LIN {X 0,Y 354.82,Z 335.287,A -85,B 0,C 180,E1 -13355.7,E2 -13355.7} C_VEL
LIN {X 0,Y 354.766,Z 335.295,A -85,B 0,C 180,E1 -13359.413,E2 -13359.413} C_VEL
LIN {X 0,Y 354.779,Z 335.292,A -85,B 0,C 180,E1 -13362.866,E2 -13362.866} C_VEL
LIN {X 0,Y 354.841,Z 335.416,A -85,B 0,C 180,E1 -13366.284,E2 -13366.284} C_VEL
LIN {X 0,Y 355.568,Z 339.552,A -85,B 0,C 180,E1 -13369.288,E2 -13369.288} C_VEL
LIN {X 0,Y 356.215,Z 343.93,A -85,B 0,C 180,E1 -13372.294,E2 -13372.294} C_VEL
LIN {X 0,Y 356.345,Z 348.318,A -85,B 0,C 180,E1 -13375.114,E2 -13375.114} C_VEL
LIN {X 0,Y 355.9,Z 353.266,A -85,B 0,C 180,E1 -13378.117,E2 -13378.117} C_VEL
LIN {X 0,Y 355.284,Z 359.294,A -85,B 0,C 180,E1 -13381.657,E2 -13381.657} C_VEL
LIN {X 0,Y 354.717,Z 365.813,A -85,B 0,C 180,E1 -13385.413,E2 -13385.413} C_VEL
LIN {X 0,Y 354.237,Z 372.787,A -85,B 0,C 180,E1 -13389.381,E2 -13389.381} C_VEL
LIN {X 0,Y 354.223,Z 372.987,A -85,B 0,C 180,E1 -13389.494,E2 -13389.494} C_VEL
LIN {X 0,Y 357.148,Z 387.433,A -85,B 0,C 180,E1 -13390.215,E2 -13390.215} C_VEL
LIN {X 0,Y 359.09,Z 400.479,A -85,B 0,C 180,E1 -13391.066,E2 -13391.066} C_VEL
LIN {X 0,Y 360.005,Z 409.631,A -85,B 0,C 180,E1 -13391.799,E2 -13391.799} C_VEL
LIN {X 0,Y 358.951,Z 420.65,A -85,B 0,C 180,E1 -13392.774,E2 -13392.774} C_VEL
LIN {X 0,Y 357.794,Z 431.905,A -85,B 0,C 180,E1 -13394.038,E2 -13394.038} C_VEL
LIN {X 0,Y 356.687,Z 441.874,A -85,B 0,C 180,E1 -13395.45,E2 -13395.45} C_VEL
LIN {X 0,Y 355.611,Z 451.544,A -85,B 0,C 180,E1 -13397.154,E2 -13397.154} C_VEL
LIN {X 0,Y 354.701,Z 459.242,A -85,B 0,C 180,E1 -13398.861,E2 -13398.861} C_VEL
LIN {X 0,Y 353.989,Z 466.343,A -85,B 0,C 180,E1 -13400.861,E2 -13400.861} C_VEL
LIN {X 0,Y 353.617,Z 471.071,A -85,B 0,C 180,E1 -13402.577,E2 -13402.577} C_VEL
LIN {X 0,Y 353.338,Z 474.682,A -85,B 0,C 180,E1 -13404.292,E2 -13404.292} C_VEL
LIN {X 0,Y 353.3,Z 476.548,A -85,B 0,C 180,E1 -13405.436,E2 -13405.436} C_VEL
LIN {X 0,Y 353.226,Z 477.946,A -85,B 0,C 180,E1 -13406.578,E2 -13406.578} C_VEL
LIN {X 0,Y 353.194,Z 479.554,A -85,B 0,C 180,E1 -13408.859,E2 -13408.859} C_VEL
LIN {X 0,Y 353.218,Z 479.771,A -85,B 0,C 180,E1 -13409.999,E2 -13409.999} C_VEL
LIN {X 0,Y 353.194,Z 479.553,A -85,B 0,C 180,E1 -13411.14,E2 -13411.14} C_VEL
LIN {X 0,Y 353.225,Z 477.945,A -85,B 0,C 180,E1 -13413.421,E2 -13413.421} C_VEL
LIN {X 0,Y 353.299,Z 476.546,A -85,B 0,C 180,E1 -13414.563,E2 -13414.563} C_VEL
LIN {X 0,Y 353.388,Z 473.979,A -85,B 0,C 180,E1 -13416.079,E2 -13416.079} C_VEL
LIN {X 0,Y 353.694,Z 469.623,A -85,B 0,C 180,E1 -13417.995,E2 -13417.995} C_VEL
LIN {X 0,Y 354.271,Z 463.506,A -85,B 0,C 180,E1 -13419.995,E2 -13419.995} C_VEL
LIN {X 0,Y 354.957,Z 456.823,A -85,B 0,C 180,E1 -13421.709,E2 -13421.709} C_VEL
LIN {X 0,Y 355.974,Z 448.538,A -85,B 0,C 180,E1 -13423.413,E2 -13423.413} C_VEL
LIN {X 0,Y 356.928,Z 440.045,A -85,B 0,C 180,E1 -13424.83,E2 -13424.83} C_VEL
LIN {X 0,Y 357.971,Z 429.549,A -85,B 0,C 180,E1 -13426.246,E2 -13426.246} C_VEL
LIN {X 0,Y 359.253,Z 417.743,A -85,B 0,C 180,E1 -13427.503,E2 -13427.503} C_VEL
LIN {X 0,Y 359.988,Z 408.468,A -85,B 0,C 180,E1 -13428.292,E2 -13428.292} C_VEL
LIN {X 0,Y 358.547,Z 396.566,A -85,B 0,C 180,E1 -13429.209,E2 -13429.209} C_VEL
LIN {X 0,Y 356.404,Z 383.633,A -85,B 0,C 180,E1 -13429.988,E2 -13429.988} C_VEL
LIN {X 0,Y 354.221,Z 372.993,A -85,B 0,C 180,E1 -13430.495,E2 -13430.495} C_VEL
LIN {X 0,Y 354.745,Z 365.803,A -85,B 0,C 180,E1 -13434.584,E2 -13434.584} C_VEL
LIN {X 0,Y 355.28,Z 359.281,A -85,B 0,C 180,E1 -13438.342,E2 -13438.342} C_VEL
LIN {X 0,Y 355.955,Z 352.692,A -85,B 0,C 180,E1 -13442.213,E2 -13442.213} C_VEL
LIN {X 0,Y 356.359,Z 348.294,A -85,B 0,C 180,E1 -13444.883,E2 -13444.883} C_VEL
LIN {X 0,Y 356.219,Z 343.604,A -85,B 0,C 180,E1 -13447.891,E2 -13447.891} C_VEL
LIN {X 0,Y 355.485,Z 338.678,A -85,B 0,C 180,E1 -13451.3,E2 -13451.3} C_VEL
LIN {X 0,Y 354.865,Z 335.288,A -85,B 0,C 180,E1 -13453.879,E2 -13453.879} C_VEL
LIN {X 0,Y 354.783,Z 335.289,A -85,B 0,C 180,E1 -13457.661,E2 -13457.661} C_VEL
LIN {X 0,Y 354.778,Z 335.295,A -85,B 0,C 180,E1 -13460.661,E2 -13460.661} C_VEL
LIN {X 0,Y 354.815,Z 335.287,A -85,B 0,C 180,E1 -13464.3,E2 -13464.3} C_VEL
LIN {X 0,Y 354.779,Z 335.289,A -85,B 0,C 180,E1 -13467.666,E2 -13467.666} C_VEL
LIN {X 0,Y 354.792,Z 335.288,A -85,B 0,C 180,E1 -13471.614,E2 -13471.614} C_VEL
LIN {X 0,Y 354.826,Z 335.284,A -85,B 0,C 180,E1 -13475.656,E2 -13475.656} C_VEL
LIN {X 0,Y 354.818,Z 335.284,A -85,B 0,C 180,E1 -13479.113,E2 -13479.113} C_VEL
LIN {X 0,Y 354.889,Z 335.276,A -85,B 0,C 180,E1 -13482.719,E2 -13482.719} C_VEL
LIN {X 0,Y 354.942,Z 335.273,A -85,B 0,C 180,E1 -13486.255,E2 -13486.255} C_VEL
LIN {X 0,Y 354.968,Z 335.269,A -85,B 0,C 180,E1 -13489.736,E2 -13489.736} C_VEL
LIN {X 0,Y 355.105,Z 335.253,A -85,B 0,C 180,E1 -13492.037,E2 -13492.037} C_VEL
LIN {X 0,Y 355.089,Z 335.252,A -85,B 0,C 180,E1 -13494.321,E2 -13494.321} C_VEL
LIN {X 0,Y 355.236,Z 335.238,A -85,B 0,C 180,E1 -13497.732,E2 -13497.732} C_VEL
LIN {X 0,Y 355.302,Z 335.227,A -85,B 0,C 180,E1 -13500,E2 -13500} C_VEL
LIN {X 0,Y 355.234,Z 335.233,A -85,B 0,C 180,E1 -13502.268,E2 -13502.268} C_VEL
LIN {X 0,Y 355.129,Z 335.246,A -85,B 0,C 180,E1 -13506.819,E2 -13506.819} C_VEL
LIN {X 0,Y 355.006,Z 335.263,A -85,B 0,C 180,E1 -13509.113,E2 -13509.113} C_VEL
LIN {X 0,Y 354.912,Z 335.273,A -85,B 0,C 180,E1 -13512.581,E2 -13512.581} C_VEL
LIN {X 0,Y 354.88,Z 335.276,A -85,B 0,C 180,E1 -13516.097,E2 -13516.097} C_VEL
LIN {X 0,Y 354.893,Z 335.275,A -85,B 0,C 180,E1 -13518.473,E2 -13518.473} C_VEL
LIN {X 0,Y 354.822,Z 335.283,A -85,B 0,C 180,E1 -13522.107,E2 -13522.107} C_VEL
LIN {X 0,Y 354.807,Z 335.286,A -85,B 0,C 180,E1 -13525.835,E2 -13525.835} C_VEL
LIN {X 0,Y 354.789,Z 335.288,A -85,B 0,C 180,E1 -13529.685,E2 -13529.685} C_VEL
LIN {X 0,Y 354.78,Z 335.29,A -85,B 0,C 180,E1 -13532.334,E2 -13532.334} C_VEL
LIN {X 0,Y 354.815,Z 335.284,A -85,B 0,C 180,E1 -13535.7,E2 -13535.7} C_VEL
LIN {X 0,Y 354.762,Z 335.291,A -85,B 0,C 180,E1 -13539.413,E2 -13539.413} C_VEL
LIN {X 0,Y 354.779,Z 335.292,A -85,B 0,C 180,E1 -13542.868,E2 -13542.868} C_VEL
LIN {X 0,Y 354.771,Z 335.293,A -85,B 0,C 180,E1 -13546.106,E2 -13546.106} C_VEL
LIN {X 0,Y 354.821,Z 335.284,A -85,B 0,C 180,E1 -13549.185,E2 -13549.185} C_VEL
LIN {X 0,Y 354.775,Z 335.296,A -85,B 0,C 180,E1 -13552.41,E2 -13552.41} C_VEL
LIN {X 0,Y 354.745,Z 335.624,A -85,B 0,C 180,E1 -13553.536,E2 -13553.536} C_VEL
LIN {X 0,Y 354.755,Z 338.537,A -85,B 0,C 180,E1 -13556.311,E2 -13556.311} C_VEL
LIN {X 0,Y 354.589,Z 341.488,A -85,B 0,C 180,E1 -13558.982,E2 -13558.982} C_VEL
LIN {X 0,Y 354.382,Z 344.409,A -85,B 0,C 180,E1 -13561.579,E2 -13561.579} C_VEL
LIN {X 0,Y 354.195,Z 347.361,A -85,B 0,C 180,E1 -13564.119,E2 -13564.119} C_VEL
LIN {X 0,Y 354.058,Z 350.336,A -85,B 0,C 180,E1 -13566.61,E2 -13566.61} C_VEL
LIN {X 0,Y 353.917,Z 354.113,A -85,B 0,C 180,E1 -13569.579,E2 -13569.579} C_VEL
LIN {X 0,Y 357.383,Z 367.353,A -85,B 0,C 180,E1 -13570.301,E2 -13570.301} C_VEL
LIN {X 0,Y 360.021,Z 379.994,A -85,B 0,C 180,E1 -13571.183,E2 -13571.183} C_VEL
LIN {X 0,Y 360.821,Z 385.123,A -85,B 0,C 180,E1 -13571.598,E2 -13571.598} C_VEL
LIN {X 0,Y 359.833,Z 396.447,A -85,B 0,C 180,E1 -13572.526,E2 -13572.526} C_VEL
LIN {X 0,Y 358.761,Z 407.702,A -85,B 0,C 180,E1 -13573.719,E2 -13573.719} C_VEL
LIN {X 0,Y 357.883,Z 416.823,A -85,B 0,C 180,E1 -13574.919,E2 -13574.919} C_VEL
LIN {X 0,Y 356.769,Z 425.661,A -85,B 0,C 180,E1 -13576.327,E2 -13576.327} C_VEL
LIN {X 0,Y 355.762,Z 434.277,A -85,B 0,C 180,E1 -13578.029,E2 -13578.029} C_VEL
LIN {X 0,Y 354.929,Z 441.145,A -85,B 0,C 180,E1 -13579.735,E2 -13579.735} C_VEL
LIN {X 0,Y 354.244,Z 446.645,A -85,B 0,C 180,E1 -13581.444,E2 -13581.444} C_VEL
LIN {X 0,Y 353.809,Z 451.294,A -85,B 0,C 180,E1 -13583.312,E2 -13583.312} C_VEL
LIN {X 0,Y 353.502,Z 455.095,A -85,B 0,C 180,E1 -13585.439,E2 -13585.439} C_VEL
LIN {X 0,Y 353.343,Z 456.494,A -85,B 0,C 180,E1 -13586.58,E2 -13586.58} C_VEL
LIN {X 0,Y 353.271,Z 458.097,A -85,B 0,C 180,E1 -13588.861,E2 -13588.861} C_VEL
LIN {X 0,Y 353.266,Z 458.329,A -85,B 0,C 180,E1 -13590.001,E2 -13590.001} C_VEL
LIN {X 0,Y 353.271,Z 458.139,A -85,B 0,C 180,E1 -13591.14,E2 -13591.14} C_VEL
LIN {X 0,Y 353.341,Z 456.589,A -85,B 0,C 180,E1 -13593.421,E2 -13593.421} C_VEL
LIN {X 0,Y 353.499,Z 455.231,A -85,B 0,C 180,E1 -13594.562,E2 -13594.562} C_VEL
LIN {X 0,Y 353.749,Z 452.388,A -85,B 0,C 180,E1 -13596.262,E2 -13596.262} C_VEL
LIN {X 0,Y 354.072,Z 448.483,A -85,B 0,C 180,E1 -13597.987,E2 -13597.987} C_VEL
LIN {X 0,Y 354.642,Z 443.469,A -85,B 0,C 180,E1 -13599.698,E2 -13599.698} C_VEL
LIN {X 0,Y 355.378,Z 437.156,A -85,B 0,C 180,E1 -13601.406,E2 -13601.406} C_VEL
LIN {X 0,Y 356.349,Z 429.251,A -85,B 0,C 180,E1 -13603.109,E2 -13603.109} C_VEL
LIN {X 0,Y 357.586,Z 419.416,A -85,B 0,C 180,E1 -13604.804,E2 -13604.804} C_VEL
LIN {X 0,Y 358.586,Z 409.357,A -85,B 0,C 180,E1 -13606.185,E2 -13606.185} C_VEL
LIN {X 0,Y 359.604,Z 398.868,A -85,B 0,C 180,E1 -13607.34,E2 -13607.34} C_VEL
LIN {X 0,Y 360.695,Z 387.231,A -85,B 0,C 180,E1 -13608.349,E2 -13608.349} C_VEL
LIN {X 0,Y 360.661,Z 383.615,A -85,B 0,C 180,E1 -13608.626,E2 -13608.626} C_VEL
LIN {X 0,Y 358.538,Z 372.554,A -85,B 0,C 180,E1 -13609.465,E2 -13609.465} C_VEL
LIN {X 0,Y 355.39,Z 359.719,A -85,B 0,C 180,E1 -13610.251,E2 -13610.251} C_VEL
LIN {X 0,Y 353.911,Z 353.989,A -85,B 0,C 180,E1 -13610.555,E2 -13610.555} C_VEL
LIN {X 0,Y 354.113,Z 348.985,A -85,B 0,C 180,E1 -13614.632,E2 -13614.632} C_VEL
LIN {X 0,Y 354.299,Z 346.026,A -85,B 0,C 180,E1 -13617.144,E2 -13617.144} C_VEL
LIN {X 0,Y 354.588,Z 341.593,A -85,B 0,C 180,E1 -13621.019,E2 -13621.019} C_VEL
LIN {X 0,Y 354.758,Z 338.678,A -85,B 0,C 180,E1 -13623.69,E2 -13623.69} C_VEL
LIN {X 0,Y 354.749,Z 335.746,A -85,B 0,C 180,E1 -13626.465,E2 -13626.465} C_VEL
LIN {X 0,Y 354.785,Z 335.294,A -85,B 0,C 180,E1 -13627.868,E2 -13627.868} C_VEL
LIN {X 0,Y 354.143,Z 335.374,A -85,B 0,C 180,E1 -13628.815,E2 -13628.815} C_VEL
LIN {X 0,Y 351.27,Z 335.728,A -85,B 0,C 180,E1 -13630.354,E2 -13630.354} C_VEL
LIN {X 0,Y 348.826,Z 336.037,A -85,B 0,C 180,E1 -13631.6,E2 -13631.6} C_VEL
LIN {X 0,Y 347.786,Z 336.161,A -85,B 0,C 180,E1 -13632.564,E2 -13632.564} C_VEL
LIN {X 0,Y 347.709,Z 336.171,A -85,B 0,C 180,E1 -13632.891,E2 -13632.891} C_VEL
LIN {X 0,Y 347.721,Z 336.169,A -85,B 0,C 180,E1 -13636.687,E2 -13636.687} C_VEL
LIN {X 0,Y 347.699,Z 336.171,A -85,B 0,C 180,E1 -13640.182,E2 -13640.182} C_VEL
LIN {X 0,Y 347.755,Z 336.164,A -85,B 0,C 180,E1 -13642.678,E2 -13642.678} C_VEL
LIN {X 0,Y 347.747,Z 336.166,A -85,B 0,C 180,E1 -13645.956,E2 -13645.956} C_VEL
LIN {X 0,Y 347.736,Z 336.168,A -85,B 0,C 180,E1 -13649.651,E2 -13649.651} C_VEL
LIN {X 0,Y 347.746,Z 336.166,A -85,B 0,C 180,E1 -13653.601,E2 -13653.601} C_VEL
LIN {X 0,Y 347.767,Z 336.162,A -85,B 0,C 180,E1 -13656.16,E2 -13656.16} C_VEL
LIN {X 0,Y 347.804,Z 336.158,A -85,B 0,C 180,E1 -13659.909,E2 -13659.909} C_VEL
LIN {X 0,Y 347.863,Z 336.152,A -85,B 0,C 180,E1 -13662.359,E2 -13662.359} C_VEL
LIN {X 0,Y 347.895,Z 336.147,A -85,B 0,C 180,E1 -13665.971,E2 -13665.971} C_VEL
LIN {X 0,Y 347.925,Z 336.143,A -85,B 0,C 180,E1 -13669.525,E2 -13669.525} C_VEL
LIN {X 0,Y 348.105,Z 336.122,A -85,B 0,C 180,E1 -13673.042,E2 -13673.042} C_VEL
LIN {X 0,Y 348.202,Z 336.109,A -85,B 0,C 180,E1 -13677.686,E2 -13677.686} C_VEL
LIN {X 0,Y 348.258,Z 336.104,A -85,B 0,C 180,E1 -13680,E2 -13680} C_VEL
LIN {X 0,Y 348.202,Z 336.114,A -85,B 0,C 180,E1 -13682.313,E2 -13682.313} C_VEL
LIN {X 0,Y 348.089,Z 336.123,A -85,B 0,C 180,E1 -13686.958,E2 -13686.958} C_VEL
LIN {X 0,Y 347.925,Z 336.145,A -85,B 0,C 180,E1 -13690.474,E2 -13690.474} C_VEL
LIN {X 0,Y 347.896,Z 336.151,A -85,B 0,C 180,E1 -13694.15,E2 -13694.15} C_VEL
LIN {X 0,Y 347.888,Z 336.15,A -85,B 0,C 180,E1 -13698.29,E2 -13698.29} C_VEL
LIN {X 0,Y 347.773,Z 336.167,A -85,B 0,C 180,E1 -13701.63,E2 -13701.63} C_VEL
LIN {X 0,Y 347.766,Z 336.164,A -85,B 0,C 180,E1 -13705.112,E2 -13705.112} C_VEL
LIN {X 0,Y 347.734,Z 336.172,A -85,B 0,C 180,E1 -13707.701,E2 -13707.701} C_VEL
LIN {X 0,Y 347.736,Z 336.167,A -85,B 0,C 180,E1 -13710.349,E2 -13710.349} C_VEL
LIN {X 0,Y 347.747,Z 336.166,A -85,B 0,C 180,E1 -13714.044,E2 -13714.044} C_VEL
LIN {X 0,Y 347.755,Z 336.17,A -85,B 0,C 180,E1 -13717.322,E2 -13717.322} C_VEL
LIN {X 0,Y 347.736,Z 336.169,A -85,B 0,C 180,E1 -13721.601,E2 -13721.601} C_VEL
LIN {X 0,Y 347.722,Z 336.173,A -85,B 0,C 180,E1 -13725.431,E2 -13725.431} C_VEL
LIN {X 0,Y 347.746,Z 336.196,A -85,B 0,C 180,E1 -13725.836,E2 -13725.836} C_VEL
LIN {X 0,Y 348.543,Z 340.513,A -85,B 0,C 180,E1 -13729.07,E2 -13729.07} C_VEL
LIN {X 0,Y 349.123,Z 344.279,A -85,B 0,C 180,E1 -13731.729,E2 -13731.729} C_VEL
LIN {X 0,Y 349.343,Z 348.156,A -85,B 0,C 180,E1 -13734.309,E2 -13734.309} C_VEL
LIN {X 0,Y 349.062,Z 352.543,A -85,B 0,C 180,E1 -13737.07,E2 -13737.07} C_VEL
LIN {X 0,Y 348.484,Z 357.61,A -85,B 0,C 180,E1 -13740.135,E2 -13740.135} C_VEL
LIN {X 0,Y 347.913,Z 363.445,A -85,B 0,C 180,E1 -13743.614,E2 -13743.614} C_VEL
LIN {X 0,Y 347.384,Z 369.908,A -85,B 0,C 180,E1 -13747.394,E2 -13747.394} C_VEL
LIN {X 0,Y 347.233,Z 372.918,A -85,B 0,C 180,E1 -13749.081,E2 -13749.081} C_VEL
LIN {X 0,Y 349.979,Z 386.18,A -85,B 0,C 180,E1 -13749.741,E2 -13749.741} C_VEL
LIN {X 0,Y 352.067,Z 399.457,A -85,B 0,C 180,E1 -13750.62,E2 -13750.62} C_VEL
LIN {X 0,Y 353.173,Z 409.418,A -85,B 0,C 180,E1 -13751.434,E2 -13751.434} C_VEL
LIN {X 0,Y 352.175,Z 420.438,A -85,B 0,C 180,E1 -13752.432,E2 -13752.432} C_VEL
LIN {X 0,Y 350.947,Z 431.692,A -85,B 0,C 180,E1 -13753.718,E2 -13753.718} C_VEL
LIN {X 0,Y 349.806,Z 441.661,A -85,B 0,C 180,E1 -13755.157,E2 -13755.157} C_VEL
LIN {X 0,Y 348.654,Z 451.33,A -85,B 0,C 180,E1 -13756.893,E2 -13756.893} C_VEL
LIN {X 0,Y 347.698,Z 459.027,A -85,B 0,C 180,E1 -13758.634,E2 -13758.634} C_VEL
LIN {X 0,Y 346.95,Z 466.128,A -85,B 0,C 180,E1 -13760.674,E2 -13760.674} C_VEL
LIN {X 0,Y 346.542,Z 470.855,A -85,B 0,C 180,E1 -13762.425,E2 -13762.425} C_VEL
LIN {X 0,Y 346.27,Z 474.467,A -85,B 0,C 180,E1 -13764.175,E2 -13764.175} C_VEL
LIN {X 0,Y 346.216,Z 476.333,A -85,B 0,C 180,E1 -13765.342,E2 -13765.342} C_VEL
LIN {X 0,Y 346.15,Z 477.731,A -85,B 0,C 180,E1 -13766.508,E2 -13766.508} C_VEL
LIN {X 0,Y 346.095,Z 479.338,A -85,B 0,C 180,E1 -13768.836,E2 -13768.836} C_VEL
LIN {X 0,Y 346.121,Z 479.556,A -85,B 0,C 180,E1 -13769.999,E2 -13769.999} C_VEL
LIN {X 0,Y 346.095,Z 479.337,A -85,B 0,C 180,E1 -13771.163,E2 -13771.163} C_VEL
LIN {X 0,Y 346.15,Z 477.73,A -85,B 0,C 180,E1 -13773.491,E2 -13773.491} C_VEL
LIN {X 0,Y 346.215,Z 476.33,A -85,B 0,C 180,E1 -13774.657,E2 -13774.657} C_VEL
LIN {X 0,Y 346.279,Z 474.111,A -85,B 0,C 180,E1 -13776.014,E2 -13776.014} C_VEL
LIN {X 0,Y 346.646,Z 469.406,A -85,B 0,C 180,E1 -13778.158,E2 -13778.158} C_VEL
LIN {X 0,Y 347.256,Z 463.289,A -85,B 0,C 180,E1 -13780.199,E2 -13780.199} C_VEL
LIN {X 0,Y 347.987,Z 456.606,A -85,B 0,C 180,E1 -13781.946,E2 -13781.946} C_VEL
LIN {X 0,Y 349.05,Z 448.32,A -85,B 0,C 180,E1 -13783.684,E2 -13783.684} C_VEL
LIN {X 0,Y 350.04,Z 439.826,A -85,B 0,C 180,E1 -13785.129,E2 -13785.129} C_VEL
LIN {X 0,Y 351.127,Z 429.329,A -85,B 0,C 180,E1 -13786.571,E2 -13786.571} C_VEL
LIN {X 0,Y 352.316,Z 418.952,A -85,B 0,C 180,E1 -13787.71,E2 -13787.71} C_VEL
LIN {X 0,Y 353.114,Z 409.34,A -85,B 0,C 180,E1 -13788.568,E2 -13788.568} C_VEL
LIN {X 0,Y 351.771,Z 397.659,A -85,B 0,C 180,E1 -13789.508,E2 -13789.508} C_VEL
LIN {X 0,Y 349.728,Z 385.039,A -85,B 0,C 180,E1 -13790.318,E2 -13790.318} C_VEL
LIN {X 0,Y 347.207,Z 372.784,A -85,B 0,C 180,E1 -13790.92,E2 -13790.92} C_VEL
LIN {X 0,Y 347.667,Z 366.586,A -85,B 0,C 180,E1 -13794.541,E2 -13794.541} C_VEL
LIN {X 0,Y 348.24,Z 360.184,A -85,B 0,C 180,E1 -13798.31,E2 -13798.31} C_VEL
LIN {X 0,Y 348.91,Z 353.676,A -85,B 0,C 180,E1 -13802.221,E2 -13802.221} C_VEL
LIN {X 0,Y 349.353,Z 349.215,A -85,B 0,C 180,E1 -13804.983,E2 -13804.983} C_VEL
LIN {X 0,Y 349.303,Z 345.922,A -85,B 0,C 180,E1 -13807.127,E2 -13807.127} C_VEL
LIN {X 0,Y 348.759,Z 341.553,A -85,B 0,C 180,E1 -13810.153,E2 -13810.153} C_VEL
LIN {X 0,Y 347.938,Z 336.657,A -85,B 0,C 180,E1 -13813.771,E2 -13813.771} C_VEL
LIN {X 0,Y 347.839,Z 336.164,A -85,B 0,C 180,E1 -13814.17,E2 -13814.17} C_VEL
LIN {X 0,Y 347.735,Z 336.17,A -85,B 0,C 180,E1 -13818.398,E2 -13818.398} C_VEL
LIN {X 0,Y 347.751,Z 336.17,A -85,B 0,C 180,E1 -13822.678,E2 -13822.678} C_VEL
LIN {X 0,Y 347.741,Z 336.167,A -85,B 0,C 180,E1 -13825.955,E2 -13825.955} C_VEL
LIN {X 0,Y 347.73,Z 336.167,A -85,B 0,C 180,E1 -13829.65,E2 -13829.65} C_VEL
LIN {X 0,Y 347.741,Z 336.166,A -85,B 0,C 180,E1 -13833.6,E2 -13833.6} C_VEL
LIN {X 0,Y 347.762,Z 336.168,A -85,B 0,C 180,E1 -13836.16,E2 -13836.16} C_VEL
LIN {X 0,Y 347.798,Z 336.161,A -85,B 0,C 180,E1 -13839.908,E2 -13839.908} C_VEL
LIN {X 0,Y 347.857,Z 336.155,A -85,B 0,C 180,E1 -13842.359,E2 -13842.359} C_VEL
LIN {X 0,Y 347.889,Z 336.152,A -85,B 0,C 180,E1 -13845.97,E2 -13845.97} C_VEL
LIN {X 0,Y 347.919,Z 336.145,A -85,B 0,C 180,E1 -13849.525,E2 -13849.525} C_VEL
LIN {X 0,Y 348.066,Z 336.131,A -85,B 0,C 180,E1 -13851.875,E2 -13851.875} C_VEL
LIN {X 0,Y 348.064,Z 336.128,A -85,B 0,C 180,E1 -13854.206,E2 -13854.206} C_VEL
LIN {X 0,Y 348.199,Z 336.114,A -85,B 0,C 180,E1 -13857.687,E2 -13857.687} C_VEL
LIN {X 0,Y 348.254,Z 336.105,A -85,B 0,C 180,E1 -13860,E2 -13860} C_VEL
LIN {X 0,Y 348.197,Z 336.109,A -85,B 0,C 180,E1 -13862.314,E2 -13862.314} C_VEL
LIN {X 0,Y 348.099,Z 336.122,A -85,B 0,C 180,E1 -13866.958,E2 -13866.958} C_VEL
LIN {X 0,Y 347.919,Z 336.143,A -85,B 0,C 180,E1 -13870.475,E2 -13870.475} C_VEL
LIN {X 0,Y 347.89,Z 336.147,A -85,B 0,C 180,E1 -13874.15,E2 -13874.15} C_VEL
LIN {X 0,Y 347.882,Z 336.148,A -85,B 0,C 180,E1 -13878.291,E2 -13878.291} C_VEL
LIN {X 0,Y 347.778,Z 336.162,A -85,B 0,C 180,E1 -13881.635,E2 -13881.635} C_VEL
LIN {X 0,Y 347.761,Z 336.168,A -85,B 0,C 180,E1 -13885.113,E2 -13885.113} C_VEL
LIN {X 0,Y 347.728,Z 336.168,A -85,B 0,C 180,E1 -13887.701,E2 -13887.701} C_VEL
LIN {X 0,Y 347.731,Z 336.168,A -85,B 0,C 180,E1 -13890.35,E2 -13890.35} C_VEL
LIN {X 0,Y 347.742,Z 336.166,A -85,B 0,C 180,E1 -13894.045,E2 -13894.045} C_VEL
LIN {X 0,Y 347.75,Z 336.165,A -85,B 0,C 180,E1 -13897.322,E2 -13897.322} C_VEL
LIN {X 0,Y 347.735,Z 336.166,A -85,B 0,C 180,E1 -13901.602,E2 -13901.602} C_VEL
LIN {X 0,Y 347.702,Z 336.172,A -85,B 0,C 180,E1 -13905.028,E2 -13905.028} C_VEL
LIN {X 0,Y 347.764,Z 336.169,A -85,B 0,C 180,E1 -13908.395,E2 -13908.395} C_VEL
LIN {X 0,Y 347.755,Z 336.168,A -85,B 0,C 180,E1 -13912.016,E2 -13912.016} C_VEL
LIN {X 0,Y 347.702,Z 336.177,A -85,B 0,C 180,E1 -13912.673,E2 -13912.673} C_VEL
LIN {X 0,Y 347.746,Z 337.271,A -85,B 0,C 180,E1 -13914.121,E2 -13914.121} C_VEL
LIN {X 0,Y 347.659,Z 340.184,A -85,B 0,C 180,E1 -13916.921,E2 -13916.921} C_VEL
LIN {X 0,Y 347.427,Z 344.024,A -85,B 0,C 180,E1 -13920.44,E2 -13920.44} C_VEL
LIN {X 0,Y 347.203,Z 347.559,A -85,B 0,C 180,E1 -13923.557,E2 -13923.557} C_VEL
LIN {X 0,Y 347.06,Z 350.542,A -85,B 0,C 180,E1 -13926.11,E2 -13926.11} C_VEL
LIN {X 0,Y 346.864,Z 354.22,A -85,B 0,C 180,E1 -13929.132,E2 -13929.132} C_VEL
LIN {X 0,Y 350.573,Z 368.215,A -85,B 0,C 180,E1 -13929.933,E2 -13929.933} C_VEL
LIN {X 0,Y 353.168,Z 380.907,A -85,B 0,C 180,E1 -13930.85,E2 -13930.85} C_VEL
LIN {X 0,Y 353.995,Z 386.567,A -85,B 0,C 180,E1 -13931.323,E2 -13931.323} C_VEL
LIN {X 0,Y 352.919,Z 398.107,A -85,B 0,C 180,E1 -13932.322,E2 -13932.322} C_VEL
LIN {X 0,Y 351.892,Z 408.521,A -85,B 0,C 180,E1 -13933.468,E2 -13933.468} C_VEL
LIN {X 0,Y 351.051,Z 417.041,A -85,B 0,C 180,E1 -13934.618,E2 -13934.618} C_VEL
LIN {X 0,Y 349.889,Z 425.879,A -85,B 0,C 180,E1 -13936.053,E2 -13936.053} C_VEL
LIN {X 0,Y 348.828,Z 434.495,A -85,B 0,C 180,E1 -13937.788,E2 -13937.788} C_VEL
LIN {X 0,Y 347.957,Z 441.362,A -85,B 0,C 180,E1 -13939.527,E2 -13939.527} C_VEL
LIN {X 0,Y 347.232,Z 446.861,A -85,B 0,C 180,E1 -13941.269,E2 -13941.269} C_VEL
LIN {X 0,Y 346.731,Z 451.805,A -85,B 0,C 180,E1 -13943.315,E2 -13943.315} C_VEL
LIN {X 0,Y 346.443,Z 455.311,A -85,B 0,C 180,E1 -13945.346,E2 -13945.346} C_VEL
LIN {X 0,Y 346.267,Z 456.709,A -85,B 0,C 180,E1 -13946.51,E2 -13946.51} C_VEL
LIN {X 0,Y 346.175,Z 458.313,A -85,B 0,C 180,E1 -13948.837,E2 -13948.837} C_VEL
LIN {X 0,Y 346.17,Z 458.544,A -85,B 0,C 180,E1 -13950.001,E2 -13950.001} C_VEL
LIN {X 0,Y 346.175,Z 458.354,A -85,B 0,C 180,E1 -13951.164,E2 -13951.164} C_VEL
LIN {X 0,Y 346.266,Z 456.803,A -85,B 0,C 180,E1 -13953.491,E2 -13953.491} C_VEL
LIN {X 0,Y 346.441,Z 455.446,A -85,B 0,C 180,E1 -13954.655,E2 -13954.655} C_VEL
LIN {X 0,Y 346.795,Z 451.829,A -85,B 0,C 180,E1 -13956.774,E2 -13956.774} C_VEL
LIN {X 0,Y 347.189,Z 447.141,A -85,B 0,C 180,E1 -13958.733,E2 -13958.733} C_VEL
LIN {X 0,Y 348.023,Z 440.705,A -85,B 0,C 180,E1 -13960.766,E2 -13960.766} C_VEL
LIN {X 0,Y 348.891,Z 433.632,A -85,B 0,C 180,E1 -13962.507,E2 -13962.507} C_VEL
LIN {X 0,Y 350.062,Z 424.816,A -85,B 0,C 180,E1 -13964.237,E2 -13964.237} C_VEL
LIN {X 0,Y 351.218,Z 415.868,A -85,B 0,C 180,E1 -13965.657,E2 -13965.657} C_VEL
LIN {X 0,Y 352.132,Z 406.131,A -85,B 0,C 180,E1 -13966.927,E2 -13966.927} C_VEL
LIN {X 0,Y 353.321,Z 394.598,A -85,B 0,C 180,E1 -13968.108,E2 -13968.108} C_VEL
LIN {X 0,Y 353.957,Z 385.341,A -85,B 0,C 180,E1 -13968.877,E2 -13968.877} C_VEL
LIN {X 0,Y 351.567,Z 372.769,A -85,B 0,C 180,E1 -13969.867,E2 -13969.867} C_VEL
LIN {X 0,Y 348.465,Z 360.116,A -85,B 0,C 180,E1 -13970.665,E2 -13970.665} C_VEL
LIN {X 0,Y 346.847,Z 354.189,A -85,B 0,C 180,E1 -13971.002,E2 -13971.002} C_VEL
LIN {X 0,Y 347.041,Z 350.179,A -85,B 0,C 180,E1 -13974.313,E2 -13974.313} C_VEL
LIN {X 0,Y 347.287,Z 346.222,A -85,B 0,C 180,E1 -13977.739,E2 -13977.739} C_VEL
LIN {X 0,Y 347.603,Z 341.78,A -85,B 0,C 180,E1 -13981.714,E2 -13981.714} C_VEL
LIN {X 0,Y 347.744,Z 338.839,A -85,B 0,C 180,E1 -13984.464,E2 -13984.464} C_VEL
LIN {X 0,Y 347.758,Z 337.181,A -85,B 0,C 180,E1 -13986.062,E2 -13986.062} C_VEL
LIN {X 0,Y 347.702,Z 336.177,A -85,B 0,C 180,E1 -13987.328,E2 -13987.328} C_VEL
LIN {X 0,Y 347.732,Z 336.169,A -85,B 0,C 180,E1 -13990.297,E2 -13990.297} C_VEL
LIN {X 0,Y 347.709,Z 336.171,A -85,B 0,C 180,E1 -13992.891,E2 -13992.891} C_VEL
LIN {X 0,Y 347.069,Z 336.255,A -85,B 0,C 180,E1 -13993.858,E2 -13993.858} C_VEL
LIN {X 0,Y 344.257,Z 336.608,A -85,B 0,C 180,E1 -13995.432,E2 -13995.432} C_VEL
LIN {X 0,Y 341.844,Z 336.908,A -85,B 0,C 180,E1 -13996.706,E2 -13996.706} C_VEL
LIN {X 0,Y 340.784,Z 337.037,A -85,B 0,C 180,E1 -13997.691,E2 -13997.691} C_VEL
LIN {X 0,Y 340.684,Z 337.046,A -85,B 0,C 180,E1 -13998.025,E2 -13998.025} C_VEL
LIN {X 0,Y 340.718,Z 337.043,A -85,B 0,C 180,E1 -14001.77,E2 -14001.77} C_VEL
LIN {X 0,Y 340.722,Z 337.043,A -85,B 0,C 180,E1 -14005.595,E2 -14005.595} C_VEL
LIN {X 0,Y 340.691,Z 337.047,A -85,B 0,C 180,E1 -14008.954,E2 -14008.954} C_VEL
LIN {X 0,Y 340.717,Z 337.046,A -85,B 0,C 180,E1 -14013.012,E2 -14013.012} C_VEL
LIN {X 0,Y 340.739,Z 337.039,A -85,B 0,C 180,E1 -14015.637,E2 -14015.637} C_VEL
LIN {X 0,Y 340.732,Z 337.04,A -85,B 0,C 180,E1 -14019.473,E2 -14019.473} C_VEL
LIN {X 0,Y 340.855,Z 337.024,A -85,B 0,C 180,E1 -14021.984,E2 -14021.984} C_VEL
LIN {X 0,Y 340.867,Z 337.022,A -85,B 0,C 180,E1 -14025.705,E2 -14025.705} C_VEL
LIN {X 0,Y 340.868,Z 337.023,A -85,B 0,C 180,E1 -14029.306,E2 -14029.306} C_VEL
LIN {X 0,Y 341.075,Z 336.999,A -85,B 0,C 180,E1 -14032.898,E2 -14032.898} C_VEL
LIN {X 0,Y 341.164,Z 336.985,A -85,B 0,C 180,E1 -14037.639,E2 -14037.639} C_VEL
LIN {X 0,Y 341.211,Z 336.982,A -85,B 0,C 180,E1 -14040,E2 -14040} C_VEL
LIN {X 0,Y 341.163,Z 336.99,A -85,B 0,C 180,E1 -14042.361,E2 -14042.361} C_VEL
LIN {X 0,Y 341.057,Z 336.999,A -85,B 0,C 180,E1 -14047.102,E2 -14047.102} C_VEL
LIN {X 0,Y 340.868,Z 337.023,A -85,B 0,C 180,E1 -14050.694,E2 -14050.694} C_VEL
LIN {X 0,Y 340.86,Z 337.026,A -85,B 0,C 180,E1 -14054.325,E2 -14054.325} C_VEL
LIN {X 0,Y 340.834,Z 337.027,A -85,B 0,C 180,E1 -14058.466,E2 -14058.466} C_VEL
LIN {X 0,Y 340.718,Z 337.046,A -85,B 0,C 180,E1 -14061.843,E2 -14061.843} C_VEL
LIN {X 0,Y 340.717,Z 337.046,A -85,B 0,C 180,E1 -14065.669,E2 -14065.669} C_VEL
LIN {X 0,Y 340.703,Z 337.048,A -85,B 0,C 180,E1 -14069.674,E2 -14069.674} C_VEL
LIN {X 0,Y 340.684,Z 337.045,A -85,B 0,C 180,E1 -14072.436,E2 -14072.436} C_VEL
LIN {X 0,Y 340.716,Z 337.047,A -85,B 0,C 180,E1 -14075.279,E2 -14075.279} C_VEL
LIN {X 0,Y 340.692,Z 337.045,A -85,B 0,C 180,E1 -14078.383,E2 -14078.383} C_VEL
LIN {X 0,Y 340.689,Z 337.045,A -85,B 0,C 180,E1 -14082.044,E2 -14082.044} C_VEL
LIN {X 0,Y 340.71,Z 337.085,A -85,B 0,C 180,E1 -14085.466,E2 -14085.466} C_VEL
LIN {X 0,Y 341.493,Z 341.448,A -85,B 0,C 180,E1 -14088.81,E2 -14088.81} C_VEL
LIN {X 0,Y 342.148,Z 345.822,A -85,B 0,C 180,E1 -14091.959,E2 -14091.959} C_VEL
LIN {X 0,Y 342.328,Z 350.201,A -85,B 0,C 180,E1 -14094.912,E2 -14094.912} C_VEL
LIN {X 0,Y 341.774,Z 355.666,A -85,B 0,C 180,E1 -14098.375,E2 -14098.375} C_VEL
LIN {X 0,Y 341.059,Z 362.18,A -85,B 0,C 180,E1 -14102.384,E2 -14102.384} C_VEL
LIN {X 0,Y 340.449,Z 368.636,A -85,B 0,C 180,E1 -14106.263,E2 -14106.263} C_VEL
LIN {X 0,Y 340.192,Z 372.777,A -85,B 0,C 180,E1 -14108.629,E2 -14108.629} C_VEL
LIN {X 0,Y 342.938,Z 385.687,A -85,B 0,C 180,E1 -14109.292,E2 -14109.292} C_VEL
LIN {X 0,Y 344.93,Z 398.233,A -85,B 0,C 180,E1 -14110.134,E2 -14110.134} C_VEL
LIN {X 0,Y 346.188,Z 409.199,A -85,B 0,C 180,E1 -14111.045,E2 -14111.045} C_VEL
LIN {X 0,Y 345.902,Z 415.833,A -85,B 0,C 180,E1 -14111.643,E2 -14111.643} C_VEL
LIN {X 0,Y 344.648,Z 426.811,A -85,B 0,C 180,E1 -14112.801,E2 -14112.801} C_VEL
LIN {X 0,Y 343.44,Z 437.284,A -85,B 0,C 180,E1 -14114.203,E2 -14114.203} C_VEL
LIN {X 0,Y 342.284,Z 446.548,A -85,B 0,C 180,E1 -14115.736,E2 -14115.736} C_VEL
LIN {X 0,Y 341.146,Z 455.176,A -85,B 0,C 180,E1 -14117.507,E2 -14117.507} C_VEL
LIN {X 0,Y 340.359,Z 462.078,A -85,B 0,C 180,E1 -14119.29,E2 -14119.29} C_VEL
LIN {X 0,Y 339.741,Z 467.611,A -85,B 0,C 180,E1 -14121.074,E2 -14121.074} C_VEL
LIN {X 0,Y 339.367,Z 471.953,A -85,B 0,C 180,E1 -14122.862,E2 -14122.862} C_VEL
LIN {X 0,Y 339.19,Z 474.252,A -85,B 0,C 180,E1 -14124.053,E2 -14124.053} C_VEL
LIN {X 0,Y 339.118,Z 476.118,A -85,B 0,C 180,E1 -14125.244,E2 -14125.244} C_VEL
LIN {X 0,Y 339.077,Z 477.517,A -85,B 0,C 180,E1 -14126.435,E2 -14126.435} C_VEL
LIN {X 0,Y 338.998,Z 479.123,A -85,B 0,C 180,E1 -14128.812,E2 -14128.812} C_VEL
LIN {X 0,Y 339.025,Z 479.34,A -85,B 0,C 180,E1 -14129.999,E2 -14129.999} C_VEL
LIN {X 0,Y 338.998,Z 479.121,A -85,B 0,C 180,E1 -14131.187,E2 -14131.187} C_VEL
LIN {X 0,Y 339.077,Z 477.514,A -85,B 0,C 180,E1 -14133.564,E2 -14133.564} C_VEL
LIN {X 0,Y 339.115,Z 476.113,A -85,B 0,C 180,E1 -14134.755,E2 -14134.755} C_VEL
LIN {X 0,Y 339.25,Z 473.169,A -85,B 0,C 180,E1 -14136.542,E2 -14136.542} C_VEL
LIN {X 0,Y 339.591,Z 469.189,A -85,B 0,C 180,E1 -14138.329,E2 -14138.329} C_VEL
LIN {X 0,Y 340.233,Z 463.07,A -85,B 0,C 180,E1 -14140.412,E2 -14140.412} C_VEL
LIN {X 0,Y 341.014,Z 456.387,A -85,B 0,C 180,E1 -14142.194,E2 -14142.194} C_VEL
LIN {X 0,Y 342.133,Z 448.102,A -85,B 0,C 180,E1 -14143.966,E2 -14143.966} C_VEL
LIN {X 0,Y 343.275,Z 438.439,A -85,B 0,C 180,E1 -14145.617,E2 -14145.617} C_VEL
LIN {X 0,Y 344.445,Z 427.932,A -85,B 0,C 180,E1 -14147.055,E2 -14147.055} C_VEL
LIN {X 0,Y 345.704,Z 417.303,A -85,B 0,C 180,E1 -14148.213,E2 -14148.213} C_VEL
LIN {X 0,Y 346.301,Z 410.893,A -85,B 0,C 180,E1 -14148.794,E2 -14148.794} C_VEL
LIN {X 0,Y 345.086,Z 399.377,A -85,B 0,C 180,E1 -14149.769,E2 -14149.769} C_VEL
LIN {X 0,Y 343.087,Z 386.647,A -85,B 0,C 180,E1 -14150.64,E2 -14150.64} C_VEL
LIN {X 0,Y 340.434,Z 374.179,A -85,B 0,C 180,E1 -14151.306,E2 -14151.306} C_VEL
LIN {X 0,Y 340.174,Z 372.483,A -85,B 0,C 180,E1 -14151.423,E2 -14151.423} C_VEL
LIN {X 0,Y 340.621,Z 366.87,A -85,B 0,C 180,E1 -14154.79,E2 -14154.79} C_VEL
LIN {X 0,Y 341.185,Z 361.086,A -85,B 0,C 180,E1 -14158.278,E2 -14158.278} C_VEL
LIN {X 0,Y 341.764,Z 355.642,A -85,B 0,C 180,E1 -14161.625,E2 -14161.625} C_VEL
LIN {X 0,Y 342.329,Z 350.153,A -85,B 0,C 180,E1 -14165.087,E2 -14165.087} C_VEL
LIN {X 0,Y 342.155,Z 345.758,A -85,B 0,C 180,E1 -14168.038,E2 -14168.038} C_VEL
LIN {X 0,Y 341.542,Z 341.398,A -85,B 0,C 180,E1 -14171.182,E2 -14171.182} C_VEL
LIN {X 0,Y 340.774,Z 337.042,A -85,B 0,C 180,E1 -14174.62,E2 -14174.62} C_VEL
LIN {X 0,Y 340.665,Z 337.053,A -85,B 0,C 180,E1 -14178.687,E2 -14178.687} C_VEL
LIN {X 0,Y 340.713,Z 337.042,A -85,B 0,C 180,E1 -14181.77,E2 -14181.77} C_VEL
LIN {X 0,Y 340.716,Z 337.041,A -85,B 0,C 180,E1 -14185.595,E2 -14185.595} C_VEL
LIN {X 0,Y 340.686,Z 337.047,A -85,B 0,C 180,E1 -14188.954,E2 -14188.954} C_VEL
LIN {X 0,Y 340.711,Z 337.043,A -85,B 0,C 180,E1 -14193.012,E2 -14193.012} C_VEL
LIN {X 0,Y 340.733,Z 337.04,A -85,B 0,C 180,E1 -14195.637,E2 -14195.637} C_VEL
LIN {X 0,Y 340.728,Z 337.04,A -85,B 0,C 180,E1 -14199.473,E2 -14199.473} C_VEL
LIN {X 0,Y 340.849,Z 337.028,A -85,B 0,C 180,E1 -14201.984,E2 -14201.984} C_VEL
LIN {X 0,Y 340.861,Z 337.025,A -85,B 0,C 180,E1 -14205.705,E2 -14205.705} C_VEL
LIN {X 0,Y 340.862,Z 337.023,A -85,B 0,C 180,E1 -14209.306,E2 -14209.306} C_VEL
LIN {X 0,Y 341.069,Z 336.997,A -85,B 0,C 180,E1 -14212.898,E2 -14212.898} C_VEL
LIN {X 0,Y 341.161,Z 336.99,A -85,B 0,C 180,E1 -14217.639,E2 -14217.639} C_VEL
LIN {X 0,Y 341.207,Z 336.983,A -85,B 0,C 180,E1 -14220,E2 -14220} C_VEL
LIN {X 0,Y 341.159,Z 336.986,A -85,B 0,C 180,E1 -14222.361,E2 -14222.361} C_VEL
LIN {X 0,Y 341.069,Z 336.999,A -85,B 0,C 180,E1 -14227.102,E2 -14227.102} C_VEL
LIN {X 0,Y 340.862,Z 337.023,A -85,B 0,C 180,E1 -14230.694,E2 -14230.694} C_VEL
LIN {X 0,Y 340.855,Z 337.023,A -85,B 0,C 180,E1 -14234.325,E2 -14234.325} C_VEL
LIN {X 0,Y 340.829,Z 337.027,A -85,B 0,C 180,E1 -14238.467,E2 -14238.467} C_VEL
LIN {X 0,Y 340.746,Z 337.037,A -85,B 0,C 180,E1 -14241.858,E2 -14241.858} C_VEL
LIN {X 0,Y 340.712,Z 337.042,A -85,B 0,C 180,E1 -14245.669,E2 -14245.669} C_VEL
LIN {X 0,Y 340.697,Z 337.044,A -85,B 0,C 180,E1 -14249.675,E2 -14249.675} C_VEL
LIN {X 0,Y 340.679,Z 337.048,A -85,B 0,C 180,E1 -14252.437,E2 -14252.437} C_VEL
LIN {X 0,Y 340.711,Z 337.043,A -85,B 0,C 180,E1 -14255.28,E2 -14255.28} C_VEL
LIN {X 0,Y 340.688,Z 337.048,A -85,B 0,C 180,E1 -14258.383,E2 -14258.383} C_VEL
LIN {X 0,Y 340.688,Z 337.046,A -85,B 0,C 180,E1 -14262.045,E2 -14262.045} C_VEL
LIN {X 0,Y 340.662,Z 337.051,A -85,B 0,C 180,E1 -14266.225,E2 -14266.225} C_VEL
LIN {X 0,Y 340.701,Z 337.047,A -85,B 0,C 180,E1 -14268.694,E2 -14268.694} C_VEL
LIN {X 0,Y 340.719,Z 337.043,A -85,B 0,C 180,E1 -14271.772,E2 -14271.772} C_VEL
LIN {X 0,Y 340.688,Z 337.742,A -85,B 0,C 180,E1 -14273.565,E2 -14273.565} C_VEL
LIN {X 0,Y 340.676,Z 340.376,A -85,B 0,C 180,E1 -14276.153,E2 -14276.153} C_VEL
LIN {X 0,Y 340.492,Z 343.308,A -85,B 0,C 180,E1 -14278.936,E2 -14278.936} C_VEL
LIN {X 0,Y 340.218,Z 347.758,A -85,B 0,C 180,E1 -14282.971,E2 -14282.971} C_VEL
LIN {X 0,Y 339.917,Z 352.277,A -85,B 0,C 180,E1 -14286.87,E2 -14286.87} C_VEL
LIN {X 0,Y 339.825,Z 354.434,A -85,B 0,C 180,E1 -14288.682,E2 -14288.682} C_VEL
LIN {X 0,Y 343.458,Z 367.939,A -85,B 0,C 180,E1 -14289.472,E2 -14289.472} C_VEL
LIN {X 0,Y 345.909,Z 379.365,A -85,B 0,C 180,E1 -14290.309,E2 -14290.309} C_VEL
LIN {X 0,Y 347.245,Z 386.933,A -85,B 0,C 180,E1 -14290.957,E2 -14290.957} C_VEL
LIN {X 0,Y 346.181,Z 398.327,A -85,B 0,C 180,E1 -14291.966,E2 -14291.966} C_VEL
LIN {X 0,Y 345.034,Z 409.324,A -85,B 0,C 180,E1 -14293.206,E2 -14293.206} C_VEL
LIN {X 0,Y 343.947,Z 419.204,A -85,B 0,C 180,E1 -14294.596,E2 -14294.596} C_VEL
LIN {X 0,Y 342.767,Z 427.694,A -85,B 0,C 180,E1 -14296.06,E2 -14296.06} C_VEL
LIN {X 0,Y 341.705,Z 435.94,A -85,B 0,C 180,E1 -14297.831,E2 -14297.831} C_VEL
LIN {X 0,Y 340.82,Z 442.582,A -85,B 0,C 180,E1 -14299.606,E2 -14299.606} C_VEL
LIN {X 0,Y 340.031,Z 448.665,A -85,B 0,C 180,E1 -14301.682,E2 -14301.682} C_VEL
LIN {X 0,Y 339.642,Z 452.351,A -85,B 0,C 180,E1 -14303.334,E2 -14303.334} C_VEL
LIN {X 0,Y 339.387,Z 455.527,A -85,B 0,C 180,E1 -14305.249,E2 -14305.249} C_VEL
LIN {X 0,Y 339.195,Z 456.925,A -85,B 0,C 180,E1 -14306.437,E2 -14306.437} C_VEL
LIN {X 0,Y 339.078,Z 458.528,A -85,B 0,C 180,E1 -14308.813,E2 -14308.813} C_VEL
LIN {X 0,Y 339.074,Z 458.76,A -85,B 0,C 180,E1 -14310.001,E2 -14310.001} C_VEL
LIN {X 0,Y 339.078,Z 458.569,A -85,B 0,C 180,E1 -14311.188,E2 -14311.188} C_VEL
LIN {X 0,Y 339.194,Z 457.018,A -85,B 0,C 180,E1 -14313.564,E2 -14313.564} C_VEL
LIN {X 0,Y 339.385,Z 455.66,A -85,B 0,C 180,E1 -14314.752,E2 -14314.752} C_VEL
LIN {X 0,Y 339.725,Z 452.313,A -85,B 0,C 180,E1 -14316.785,E2 -14316.785} C_VEL
LIN {X 0,Y 340.157,Z 447.356,A -85,B 0,C 180,E1 -14318.915,E2 -14318.915} C_VEL
LIN {X 0,Y 340.944,Z 441.922,A -85,B 0,C 180,E1 -14320.692,E2 -14320.692} C_VEL
LIN {X 0,Y 341.824,Z 435.134,A -85,B 0,C 180,E1 -14322.468,E2 -14322.468} C_VEL
LIN {X 0,Y 342.719,Z 428.199,A -85,B 0,C 180,E1 -14323.943,E2 -14323.943} C_VEL
LIN {X 0,Y 343.891,Z 419.839,A -85,B 0,C 180,E1 -14325.407,E2 -14325.407} C_VEL
LIN {X 0,Y 344.936,Z 409.962,A -85,B 0,C 180,E1 -14326.821,E2 -14326.821} C_VEL
LIN {X 0,Y 346.109,Z 399.287,A -85,B 0,C 180,E1 -14328.039,E2 -14328.039} C_VEL
LIN {X 0,Y 347.244,Z 386.938,A -85,B 0,C 180,E1 -14329.147,E2 -14329.147} C_VEL
LIN {X 0,Y 344.911,Z 374.348,A -85,B 0,C 180,E1 -14330.185,E2 -14330.185} C_VEL
LIN {X 0,Y 341.794,Z 361.548,A -85,B 0,C 180,E1 -14331.036,E2 -14331.036} C_VEL
LIN {X 0,Y 339.818,Z 354.396,A -85,B 0,C 180,E1 -14331.459,E2 -14331.459} C_VEL
LIN {X 0,Y 340.003,Z 350.71,A -85,B 0,C 180,E1 -14334.563,E2 -14334.563} C_VEL
LIN {X 0,Y 340.225,Z 347.544,A -85,B 0,C 180,E1 -14337.346,E2 -14337.346} C_VEL
LIN {X 0,Y 340.495,Z 343.428,A -85,B 0,C 180,E1 -14341.065,E2 -14341.065} C_VEL
LIN {X 0,Y 340.719,Z 339.888,A -85,B 0,C 180,E1 -14344.403,E2 -14344.403} C_VEL
LIN {X 0,Y 340.675,Z 337.527,A -85,B 0,C 180,E1 -14346.745,E2 -14346.745} C_VEL
LIN {X 0,Y 340.698,Z 337.048,A -85,B 0,C 180,E1 -14348.383,E2 -14348.383} C_VEL
LIN {X 0,Y 340.699,Z 337.046,A -85,B 0,C 180,E1 -14352.045,E2 -14352.045} C_VEL
LIN {X 0,Y 340.649,Z 337.05,A -85,B 0,C 180,E1 -14356.227,E2 -14356.227} C_VEL
LIN {X 0,Y 340.684,Z 337.046,A -85,B 0,C 180,E1 -14358.025,E2 -14358.025} C_VEL
LIN {X 0,Y 339.987,Z 337.135,A -85,B 0,C 180,E1 -14359.012,E2 -14359.012} C_VEL
LIN {X 0,Y 337.146,Z 337.49,A -85,B 0,C 180,E1 -14360.618,E2 -14360.618} C_VEL
LIN {X 0,Y 334.761,Z 337.79,A -85,B 0,C 180,E1 -14361.918,E2 -14361.918} C_VEL
LIN {X 0,Y 333.742,Z 337.915,A -85,B 0,C 180,E1 -14362.924,E2 -14362.924} C_VEL
LIN {X 0,Y 333.66,Z 337.923,A -85,B 0,C 180,E1 -14363.264,E2 -14363.264} C_VEL
LIN {X 0,Y 333.635,Z 337.925,A -85,B 0,C 180,E1 -14366.791,E2 -14366.791} C_VEL
LIN {X 0,Y 333.659,Z 337.921,A -85,B 0,C 180,E1 -14369.722,E2 -14369.722} C_VEL
LIN {X 0,Y 333.653,Z 337.921,A -85,B 0,C 180,E1 -14373.747,E2 -14373.747} C_VEL
LIN {X 0,Y 333.657,Z 337.921,A -85,B 0,C 180,E1 -14376.409,E2 -14376.409} C_VEL
LIN {X 0,Y 333.729,Z 337.912,A -85,B 0,C 180,E1 -14380.309,E2 -14380.309} C_VEL
LIN {X 0,Y 333.744,Z 337.915,A -85,B 0,C 180,E1 -14382.854,E2 -14382.854} C_VEL
LIN {X 0,Y 333.794,Z 337.908,A -85,B 0,C 180,E1 -14386.608,E2 -14386.608} C_VEL
LIN {X 0,Y 333.86,Z 337.898,A -85,B 0,C 180,E1 -14390.305,E2 -14390.305} C_VEL
LIN {X 0,Y 334.024,Z 337.878,A -85,B 0,C 180,E1 -14392.747,E2 -14392.747} C_VEL
LIN {X 0,Y 333.807,Z 337.902,A -85,B 0,C 180,E1 -14395.169,E2 -14395.169} C_VEL
LIN {X 0,Y 334.102,Z 337.865,A -85,B 0,C 180,E1 -14397.589,E2 -14397.589} C_VEL
LIN {X 0,Y 334.164,Z 337.86,A -85,B 0,C 180,E1 -14400,E2 -14400} C_VEL
LIN {X 0,Y 334.101,Z 337.869,A -85,B 0,C 180,E1 -14402.411,E2 -14402.411} C_VEL
LIN {X 0,Y 334.012,Z 337.881,A -85,B 0,C 180,E1 -14406.039,E2 -14406.039} C_VEL
LIN {X 0,Y 333.956,Z 337.886,A -85,B 0,C 180,E1 -14408.471,E2 -14408.471} C_VEL
LIN {X 0,Y 333.788,Z 337.909,A -85,B 0,C 180,E1 -14412.155,E2 -14412.155} C_VEL
LIN {X 0,Y 333.774,Z 337.911,A -85,B 0,C 180,E1 -14415.886,E2 -14415.886} C_VEL
LIN {X 0,Y 333.793,Z 337.904,A -85,B 0,C 180,E1 -14418.655,E2 -14418.655} C_VEL
LIN {X 0,Y 333.654,Z 337.922,A -85,B 0,C 180,E1 -14422.281,E2 -14422.281} C_VEL
LIN {X 0,Y 333.687,Z 337.918,A -85,B 0,C 180,E1 -14425.09,E2 -14425.09} C_VEL
LIN {X 0,Y 333.65,Z 337.923,A -85,B 0,C 180,E1 -14428.978,E2 -14428.978} C_VEL
LIN {X 0,Y 333.642,Z 337.923,A -85,B 0,C 180,E1 -14432.587,E2 -14432.587} C_VEL
LIN {X 0,Y 333.674,Z 337.919,A -85,B 0,C 180,E1 -14436.139,E2 -14436.139} C_VEL
LIN {X 0,Y 333.618,Z 337.93,A -85,B 0,C 180,E1 -14439.196,E2 -14439.196} C_VEL
LIN {X 0,Y 333.625,Z 337.926,A -85,B 0,C 180,E1 -14442.499,E2 -14442.499} C_VEL
LIN {X 0,Y 333.66,Z 338.034,A -85,B 0,C 180,E1 -14445.134,E2 -14445.134} C_VEL
LIN {X 0,Y 334.265,Z 341.293,A -85,B 0,C 180,E1 -14447.716,E2 -14447.716} C_VEL
LIN {X 0,Y 334.971,Z 345.656,A -85,B 0,C 180,E1 -14450.992,E2 -14450.992} C_VEL
LIN {X 0,Y 335.333,Z 350.03,A -85,B 0,C 180,E1 -14454.068,E2 -14454.068} C_VEL
LIN {X 0,Y 334.971,Z 354.578,A -85,B 0,C 180,E1 -14457.06,E2 -14457.06} C_VEL
LIN {X 0,Y 334.219,Z 360.896,A -85,B 0,C 180,E1 -14461.076,E2 -14461.076} C_VEL
LIN {X 0,Y 333.571,Z 367.372,A -85,B 0,C 180,E1 -14465.078,E2 -14465.078} C_VEL
LIN {X 0,Y 333.16,Z 372.491,A -85,B 0,C 180,E1 -14468.153,E2 -14468.153} C_VEL
LIN {X 0,Y 335.971,Z 385.37,A -85,B 0,C 180,E1 -14468.837,E2 -14468.837} C_VEL
LIN {X 0,Y 338.033,Z 398.017,A -85,B 0,C 180,E1 -14469.711,E2 -14469.711} C_VEL
LIN {X 0,Y 339.421,Z 410.761,A -85,B 0,C 180,E1 -14470.81,E2 -14470.81} C_VEL
LIN {X 0,Y 338.631,Z 420.015,A -85,B 0,C 180,E1 -14471.705,E2 -14471.705} C_VEL
LIN {X 0,Y 337.273,Z 431.265,A -85,B 0,C 180,E1 -14473.038,E2 -14473.038} C_VEL
LIN {X 0,Y 336.084,Z 441.235,A -85,B 0,C 180,E1 -14474.536,E2 -14474.536} C_VEL
LIN {X 0,Y 334.995,Z 449.412,A -85,B 0,C 180,E1 -14476.039,E2 -14476.039} C_VEL
LIN {X 0,Y 333.851,Z 457.435,A -85,B 0,C 180,E1 -14477.847,E2 -14477.847} C_VEL
LIN {X 0,Y 333.115,Z 463.875,A -85,B 0,C 180,E1 -14479.669,E2 -14479.669} C_VEL
LIN {X 0,Y 332.558,Z 468.99,A -85,B 0,C 180,E1 -14481.493,E2 -14481.493} C_VEL
LIN {X 0,Y 332.192,Z 472.964,A -85,B 0,C 180,E1 -14483.318,E2 -14483.318} C_VEL
LIN {X 0,Y 332.024,Z 475.902,A -85,B 0,C 180,E1 -14485.143,E2 -14485.143} C_VEL
LIN {X 0,Y 332.005,Z 477.302,A -85,B 0,C 180,E1 -14486.359,E2 -14486.359} C_VEL
LIN {X 0,Y 331.905,Z 478.908,A -85,B 0,C 180,E1 -14488.786,E2 -14488.786} C_VEL
LIN {X 0,Y 331.929,Z 479.125,A -85,B 0,C 180,E1 -14489.999,E2 -14489.999} C_VEL
LIN {X 0,Y 331.905,Z 478.906,A -85,B 0,C 180,E1 -14491.213,E2 -14491.213} C_VEL
LIN {X 0,Y 332.004,Z 477.299,A -85,B 0,C 180,E1 -14493.64,E2 -14493.64} C_VEL
LIN {X 0,Y 332.072,Z 474.344,A -85,B 0,C 180,E1 -14495.894,E2 -14495.894} C_VEL
LIN {X 0,Y 332.39,Z 470.406,A -85,B 0,C 180,E1 -14497.899,E2 -14497.899} C_VEL
LIN {X 0,Y 332.892,Z 465.676,A -85,B 0,C 180,E1 -14499.723,E2 -14499.723} C_VEL
LIN {X 0,Y 333.696,Z 458.57,A -85,B 0,C 180,E1 -14501.849,E2 -14501.849} C_VEL
LIN {X 0,Y 334.784,Z 450.865,A -85,B 0,C 180,E1 -14503.66,E2 -14503.66} C_VEL
LIN {X 0,Y 336.056,Z 441.189,A -85,B 0,C 180,E1 -14505.464,E2 -14505.464} C_VEL
LIN {X 0,Y 337.231,Z 431.207,A -85,B 0,C 180,E1 -14506.963,E2 -14506.963} C_VEL
LIN {X 0,Y 338.622,Z 419.941,A -85,B 0,C 180,E1 -14508.294,E2 -14508.294} C_VEL
LIN {X 0,Y 339.393,Z 410.666,A -85,B 0,C 180,E1 -14509.191,E2 -14509.191} C_VEL
LIN {X 0,Y 338.145,Z 399.146,A -85,B 0,C 180,E1 -14510.192,E2 -14510.192} C_VEL
LIN {X 0,Y 336.137,Z 386.433,A -85,B 0,C 180,E1 -14511.086,E2 -14511.086} C_VEL
LIN {X 0,Y 333.296,Z 373.453,A -85,B 0,C 180,E1 -14511.8,E2 -14511.8} C_VEL
LIN {X 0,Y 333.157,Z 372.311,A -85,B 0,C 180,E1 -14511.875,E2 -14511.875} C_VEL
LIN {X 0,Y 333.605,Z 367.131,A -85,B 0,C 180,E1 -14515.059,E2 -14515.059} C_VEL
LIN {X 0,Y 334.213,Z 360.894,A -85,B 0,C 180,E1 -14518.923,E2 -14518.923} C_VEL
LIN {X 0,Y 334.966,Z 354.549,A -85,B 0,C 180,E1 -14522.939,E2 -14522.939} C_VEL
LIN {X 0,Y 335.326,Z 349.985,A -85,B 0,C 180,E1 -14525.932,E2 -14525.932} C_VEL
LIN {X 0,Y 334.985,Z 345.487,A -85,B 0,C 180,E1 -14529.08,E2 -14529.08} C_VEL
LIN {X 0,Y 334.242,Z 340.81,A -85,B 0,C 180,E1 -14532.614,E2 -14532.614} C_VEL
LIN {X 0,Y 333.705,Z 337.921,A -85,B 0,C 180,E1 -14535.065,E2 -14535.065} C_VEL
LIN {X 0,Y 333.633,Z 337.925,A -85,B 0,C 180,E1 -14537.617,E2 -14537.617} C_VEL
LIN {X 0,Y 333.628,Z 337.927,A -85,B 0,C 180,E1 -14541.205,E2 -14541.205} C_VEL
LIN {X 0,Y 333.669,Z 337.92,A -85,B 0,C 180,E1 -14543.86,E2 -14543.86} C_VEL
LIN {X 0,Y 333.636,Z 337.924,A -85,B 0,C 180,E1 -14547.412,E2 -14547.412} C_VEL
LIN {X 0,Y 333.645,Z 337.924,A -85,B 0,C 180,E1 -14551.022,E2 -14551.022} C_VEL
LIN {X 0,Y 333.688,Z 337.917,A -85,B 0,C 180,E1 -14555.088,E2 -14555.088} C_VEL
LIN {X 0,Y 333.666,Z 337.92,A -85,B 0,C 180,E1 -14559.018,E2 -14559.018} C_VEL
LIN {X 0,Y 333.785,Z 337.905,A -85,B 0,C 180,E1 -14561.589,E2 -14561.589} C_VEL
LIN {X 0,Y 333.8,Z 337.904,A -85,B 0,C 180,E1 -14565.576,E2 -14565.576} C_VEL
LIN {X 0,Y 333.824,Z 337.899,A -85,B 0,C 180,E1 -14569.078,E2 -14569.078} C_VEL
LIN {X 0,Y 334.019,Z 337.875,A -85,B 0,C 180,E1 -14572.747,E2 -14572.747} C_VEL
LIN {X 0,Y 333.806,Z 337.902,A -85,B 0,C 180,E1 -14575.169,E2 -14575.169} C_VEL
LIN {X 0,Y 334.098,Z 337.869,A -85,B 0,C 180,E1 -14577.589,E2 -14577.589} C_VEL
LIN {X 0,Y 334.16,Z 337.861,A -85,B 0,C 180,E1 -14580,E2 -14580} C_VEL
LIN {X 0,Y 334.096,Z 337.865,A -85,B 0,C 180,E1 -14582.411,E2 -14582.411} C_VEL
LIN {X 0,Y 334.018,Z 337.879,A -85,B 0,C 180,E1 -14587.253,E2 -14587.253} C_VEL
LIN {X 0,Y 333.825,Z 337.901,A -85,B 0,C 180,E1 -14590.922,E2 -14590.922} C_VEL
LIN {X 0,Y 333.8,Z 337.903,A -85,B 0,C 180,E1 -14594.635,E2 -14594.635} C_VEL
LIN {X 0,Y 333.788,Z 337.905,A -85,B 0,C 180,E1 -14598.655,E2 -14598.655} C_VEL
LIN {X 0,Y 333.683,Z 337.917,A -85,B 0,C 180,E1 -14602.279,E2 -14602.279} C_VEL
LIN {X 0,Y 333.682,Z 337.923,A -85,B 0,C 180,E1 -14605.091,E2 -14605.091} C_VEL
LIN {X 0,Y 333.645,Z 337.927,A -85,B 0,C 180,E1 -14608.979,E2 -14608.979} C_VEL
LIN {X 0,Y 333.637,Z 337.926,A -85,B 0,C 180,E1 -14612.588,E2 -14612.588} C_VEL
LIN {X 0,Y 333.669,Z 337.92,A -85,B 0,C 180,E1 -14616.14,E2 -14616.14} C_VEL
LIN {X 0,Y 333.614,Z 337.927,A -85,B 0,C 180,E1 -14619.197,E2 -14619.197} C_VEL
LIN {X 0,Y 333.624,Z 337.93,A -85,B 0,C 180,E1 -14622.5,E2 -14622.5} C_VEL
LIN {X 0,Y 333.603,Z 337.929,A -85,B 0,C 180,E1 -14625.958,E2 -14625.958} C_VEL
LIN {X 0,Y 333.653,Z 337.922,A -85,B 0,C 180,E1 -14629.315,E2 -14629.315} C_VEL
LIN {X 0,Y 333.634,Z 337.929,A -85,B 0,C 180,E1 -14632.348,E2 -14632.348} C_VEL
LIN {X 0,Y 333.655,Z 339.076,A -85,B 0,C 180,E1 -14633.86,E2 -14633.86} C_VEL
LIN {X 0,Y 333.592,Z 342.03,A -85,B 0,C 180,E1 -14636.788,E2 -14636.788} C_VEL
LIN {X 0,Y 333.37,Z 345.193,A -85,B 0,C 180,E1 -14639.809,E2 -14639.809} C_VEL
LIN {X 0,Y 333.218,Z 347.955,A -85,B 0,C 180,E1 -14642.355,E2 -14642.355} C_VEL
LIN {X 0,Y 332.879,Z 352.484,A -85,B 0,C 180,E1 -14646.351,E2 -14646.351} C_VEL
LIN {X 0,Y 332.776,Z 354.644,A -85,B 0,C 180,E1 -14648.195,E2 -14648.195} C_VEL
LIN {X 0,Y 336.898,Z 369.832,A -85,B 0,C 180,E1 -14649.142,E2 -14649.142} C_VEL
LIN {X 0,Y 339.417,Z 382.055,A -85,B 0,C 180,E1 -14650.091,E2 -14650.091} C_VEL
LIN {X 0,Y 340.427,Z 388.88,A -85,B 0,C 180,E1 -14650.713,E2 -14650.713} C_VEL
LIN {X 0,Y 339.279,Z 399.969,A -85,B 0,C 180,E1 -14651.742,E2 -14651.742} C_VEL
LIN {X 0,Y 338.184,Z 410.121,A -85,B 0,C 180,E1 -14652.932,E2 -14652.932} C_VEL
LIN {X 0,Y 337.102,Z 419.423,A -85,B 0,C 180,E1 -14654.275,E2 -14654.275} C_VEL
LIN {X 0,Y 335.89,Z 427.912,A -85,B 0,C 180,E1 -14655.769,E2 -14655.769} C_VEL
LIN {X 0,Y 334.782,Z 436.157,A -85,B 0,C 180,E1 -14657.575,E2 -14657.575} C_VEL
LIN {X 0,Y 333.853,Z 442.798,A -85,B 0,C 180,E1 -14659.386,E2 -14659.386} C_VEL
LIN {X 0,Y 333.018,Z 448.882,A -85,B 0,C 180,E1 -14661.505,E2 -14661.505} C_VEL
LIN {X 0,Y 332.568,Z 452.838,A -85,B 0,C 180,E1 -14663.331,E2 -14663.331} C_VEL
LIN {X 0,Y 332.31,Z 455.743,A -85,B 0,C 180,E1 -14665.148,E2 -14665.148} C_VEL
LIN {X 0,Y 332.126,Z 457.14,A -85,B 0,C 180,E1 -14666.361,E2 -14666.361} C_VEL
LIN {X 0,Y 331.982,Z 458.744,A -85,B 0,C 180,E1 -14668.788,E2 -14668.788} C_VEL
LIN {X 0,Y 331.978,Z 458.975,A -85,B 0,C 180,E1 -14670.001,E2 -14670.001} C_VEL
LIN {X 0,Y 331.982,Z 458.784,A -85,B 0,C 180,E1 -14671.214,E2 -14671.214} C_VEL
LIN {X 0,Y 332.125,Z 457.232,A -85,B 0,C 180,E1 -14673.64,E2 -14673.64} C_VEL
LIN {X 0,Y 332.308,Z 455.875,A -85,B 0,C 180,E1 -14674.853,E2 -14674.853} C_VEL
LIN {X 0,Y 332.656,Z 452.788,A -85,B 0,C 180,E1 -14676.797,E2 -14676.797} C_VEL
LIN {X 0,Y 332.952,Z 449.127,A -85,B 0,C 180,E1 -14678.497,E2 -14678.497} C_VEL
LIN {X 0,Y 333.664,Z 444.11,A -85,B 0,C 180,E1 -14680.314,E2 -14680.314} C_VEL
LIN {X 0,Y 334.526,Z 437.796,A -85,B 0,C 180,E1 -14682.128,E2 -14682.128} C_VEL
LIN {X 0,Y 335.633,Z 429.89,A -85,B 0,C 180,E1 -14683.934,E2 -14683.934} C_VEL
LIN {X 0,Y 337.044,Z 420.052,A -85,B 0,C 180,E1 -14685.728,E2 -14685.728} C_VEL
LIN {X 0,Y 338.146,Z 410.173,A -85,B 0,C 180,E1 -14687.169,E2 -14687.169} C_VEL
LIN {X 0,Y 339.368,Z 399.497,A -85,B 0,C 180,E1 -14688.41,E2 -14688.41} C_VEL
LIN {X 0,Y 340.488,Z 388.276,A -85,B 0,C 180,E1 -14689.443,E2 -14689.443} C_VEL
LIN {X 0,Y 338.44,Z 376.814,A -85,B 0,C 180,E1 -14690.448,E2 -14690.448} C_VEL
LIN {X 0,Y 335.441,Z 364.121,A -85,B 0,C 180,E1 -14691.348,E2 -14691.348} C_VEL
LIN {X 0,Y 332.783,Z 354.653,A -85,B 0,C 180,E1 -14691.906,E2 -14691.906} C_VEL
LIN {X 0,Y 332.97,Z 351.085,A -85,B 0,C 180,E1 -14694.97,E2 -14694.97} C_VEL
LIN {X 0,Y 333.203,Z 348.103,A -85,B 0,C 180,E1 -14697.647,E2 -14697.647} C_VEL
LIN {X 0,Y 333.498,Z 343.614,A -85,B 0,C 180,E1 -14701.792,E2 -14701.792} C_VEL
LIN {X 0,Y 333.702,Z 340.533,A -85,B 0,C 180,E1 -14704.778,E2 -14704.778} C_VEL
LIN {X 0,Y 333.636,Z 337.93,A -85,B 0,C 180,E1 -14707.653,E2 -14707.653} C_VEL
LIN {X 0,Y 333.647,Z 337.923,A -85,B 0,C 180,E1 -14710.767,E2 -14710.767} C_VEL
LIN {X 0,Y 333.592,Z 337.93,A -85,B 0,C 180,E1 -14714.25,E2 -14714.25} C_VEL
LIN {X 0,Y 333.602,Z 337.929,A -85,B 0,C 180,E1 -14718.012,E2 -14718.012} C_VEL
LIN {X 0,Y 333.642,Z 337.922,A -85,B 0,C 180,E1 -14722.347,E2 -14722.347} C_VEL
LIN {X 0,Y 333.66,Z 337.923,A -85,B 0,C 180,E1 -14723.264,E2 -14723.264} C_VEL
LIN {X 0,Y 332.986,Z 338.005,A -85,B 0,C 180,E1 -14724.272,E2 -14724.272} C_VEL
LIN {X 0,Y 330.102,Z 338.364,A -85,B 0,C 180,E1 -14725.91,E2 -14725.91} C_VEL
LIN {X 0,Y 327.668,Z 338.671,A -85,B 0,C 180,E1 -14727.238,E2 -14727.238} C_VEL
LIN {X 0,Y 326.637,Z 338.795,A -85,B 0,C 180,E1 -14728.266,E2 -14728.266} C_VEL
LIN {X 0,Y 326.561,Z 338.805,A -85,B 0,C 180,E1 -14728.614,E2 -14728.614} C_VEL
LIN {X 0,Y 326.599,Z 338.8,A -85,B 0,C 180,E1 -14731.916,E2 -14731.916} C_VEL
LIN {X 0,Y 326.629,Z 338.796,A -85,B 0,C 180,E1 -14735.869,E2 -14735.869} C_VEL
LIN {X 0,Y 326.656,Z 338.792,A -85,B 0,C 180,E1 -14739.864,E2 -14739.864} C_VEL
LIN {X 0,Y 326.697,Z 338.79,A -85,B 0,C 180,E1 -14742.472,E2 -14742.472} C_VEL
LIN {X 0,Y 326.756,Z 338.782,A -85,B 0,C 180,E1 -14746.314,E2 -14746.314} C_VEL
LIN {X 0,Y 326.811,Z 338.775,A -85,B 0,C 180,E1 -14750.094,E2 -14750.094} C_VEL
LIN {X 0,Y 326.975,Z 338.758,A -85,B 0,C 180,E1 -14752.59,E2 -14752.59} C_VEL
LIN {X 0,Y 326.774,Z 338.779,A -85,B 0,C 180,E1 -14755.065,E2 -14755.065} C_VEL
LIN {X 0,Y 327.043,Z 338.744,A -85,B 0,C 180,E1 -14757.537,E2 -14757.537} C_VEL
LIN {X 0,Y 327.119,Z 338.737,A -85,B 0,C 180,E1 -14760,E2 -14760} C_VEL
LIN {X 0,Y 327.042,Z 338.748,A -85,B 0,C 180,E1 -14762.463,E2 -14762.463} C_VEL
LIN {X 0,Y 326.987,Z 338.757,A -85,B 0,C 180,E1 -14766.169,E2 -14766.169} C_VEL
LIN {X 0,Y 326.803,Z 338.779,A -85,B 0,C 180,E1 -14769.907,E2 -14769.907} C_VEL
LIN {X 0,Y 326.756,Z 338.784,A -85,B 0,C 180,E1 -14773.685,E2 -14773.685} C_VEL
LIN {X 0,Y 326.696,Z 338.791,A -85,B 0,C 180,E1 -14777.528,E2 -14777.528} C_VEL
LIN {X 0,Y 326.656,Z 338.795,A -85,B 0,C 180,E1 -14780.135,E2 -14780.135} C_VEL
LIN {X 0,Y 326.631,Z 338.798,A -85,B 0,C 180,E1 -14784.131,E2 -14784.131} C_VEL
LIN {X 0,Y 326.596,Z 338.801,A -85,B 0,C 180,E1 -14788.256,E2 -14788.256} C_VEL
LIN {X 0,Y 326.571,Z 338.806,A -85,B 0,C 180,E1 -14791.097,E2 -14791.097} C_VEL
LIN {X 0,Y 326.605,Z 338.801,A -85,B 0,C 180,E1 -14794.02,E2 -14794.02} C_VEL
LIN {X 0,Y 326.622,Z 338.802,A -85,B 0,C 180,E1 -14797.238,E2 -14797.238} C_VEL
LIN {X 0,Y 326.542,Z 338.811,A -85,B 0,C 180,E1 -14801.124,E2 -14801.124} C_VEL
LIN {X 0,Y 326.613,Z 338.953,A -85,B 0,C 180,E1 -14804.758,E2 -14804.758} C_VEL
LIN {X 0,Y 327.492,Z 343.821,A -85,B 0,C 180,E1 -14808.686,E2 -14808.686} C_VEL
LIN {X 0,Y 328.102,Z 347.669,A -85,B 0,C 180,E1 -14811.597,E2 -14811.597} C_VEL
LIN {X 0,Y 328.285,Z 352.036,A -85,B 0,C 180,E1 -14814.689,E2 -14814.689} C_VEL
LIN {X 0,Y 327.709,Z 357.477,A -85,B 0,C 180,E1 -14818.303,E2 -14818.303} C_VEL
LIN {X 0,Y 326.945,Z 363.946,A -85,B 0,C 180,E1 -14822.473,E2 -14822.473} C_VEL
LIN {X 0,Y 326.287,Z 370.336,A -85,B 0,C 180,E1 -14826.517,E2 -14826.517} C_VEL
LIN {X 0,Y 326.162,Z 372.141,A -85,B 0,C 180,E1 -14827.65,E2 -14827.65} C_VEL
LIN {X 0,Y 329.102,Z 385.608,A -85,B 0,C 180,E1 -14828.397,E2 -14828.397} C_VEL
LIN {X 0,Y 331.112,Z 397.8,A -85,B 0,C 180,E1 -14829.268,E2 -14829.268} C_VEL
LIN {X 0,Y 332.5,Z 410.543,A -85,B 0,C 180,E1 -14830.394,E2 -14830.394} C_VEL
LIN {X 0,Y 332.405,Z 415.41,A -85,B 0,C 180,E1 -14830.87,E2 -14830.87} C_VEL
LIN {X 0,Y 331.084,Z 426.386,A -85,B 0,C 180,E1 -14832.073,E2 -14832.073} C_VEL
LIN {X 0,Y 329.799,Z 436.359,A -85,B 0,C 180,E1 -14833.45,E2 -14833.45} C_VEL
LIN {X 0,Y 328.451,Z 446.119,A -85,B 0,C 180,E1 -14835.121,E2 -14835.121} C_VEL
LIN {X 0,Y 327.262,Z 454.747,A -85,B 0,C 180,E1 -14836.968,E2 -14836.968} C_VEL
LIN {X 0,Y 326.347,Z 461.648,A -85,B 0,C 180,E1 -14838.824,E2 -14838.824} C_VEL
LIN {X 0,Y 325.672,Z 467.181,A -85,B 0,C 180,E1 -14840.685,E2 -14840.685} C_VEL
LIN {X 0,Y 325.226,Z 471.522,A -85,B 0,C 180,E1 -14842.55,E2 -14842.55} C_VEL
LIN {X 0,Y 325,Z 474.364,A -85,B 0,C 180,E1 -14844.118,E2 -14844.118} C_VEL
LIN {X 0,Y 324.911,Z 477.087,A -85,B 0,C 180,E1 -14846.279,E2 -14846.279} C_VEL
LIN {X 0,Y 324.815,Z 478.693,A -85,B 0,C 180,E1 -14848.76,E2 -14848.76} C_VEL
LIN {X 0,Y 324.835,Z 478.91,A -85,B 0,C 180,E1 -14849.999,E2 -14849.999} C_VEL
LIN {X 0,Y 324.815,Z 478.691,A -85,B 0,C 180,E1 -14851.239,E2 -14851.239} C_VEL
LIN {X 0,Y 324.91,Z 477.083,A -85,B 0,C 180,E1 -14853.72,E2 -14853.72} C_VEL
LIN {X 0,Y 324.996,Z 474.363,A -85,B 0,C 180,E1 -14855.875,E2 -14855.875} C_VEL
LIN {X 0,Y 325.344,Z 470.189,A -85,B 0,C 180,E1 -14858.071,E2 -14858.071} C_VEL
LIN {X 0,Y 325.872,Z 465.458,A -85,B 0,C 180,E1 -14859.934,E2 -14859.934} C_VEL
LIN {X 0,Y 326.726,Z 458.352,A -85,B 0,C 180,E1 -14862.106,E2 -14862.106} C_VEL
LIN {X 0,Y 327.876,Z 450.647,A -85,B 0,C 180,E1 -14863.953,E2 -14863.953} C_VEL
LIN {X 0,Y 329.193,Z 440.97,A -85,B 0,C 180,E1 -14865.794,E2 -14865.794} C_VEL
LIN {X 0,Y 330.417,Z 430.987,A -85,B 0,C 180,E1 -14867.323,E2 -14867.323} C_VEL
LIN {X 0,Y 331.862,Z 419.72,A -85,B 0,C 180,E1 -14868.681,E2 -14868.681} C_VEL
LIN {X 0,Y 332.59,Z 412.143,A -85,B 0,C 180,E1 -14869.439,E2 -14869.439} C_VEL
LIN {X 0,Y 331.414,Z 400.472,A -85,B 0,C 180,E1 -14870.51,E2 -14870.51} C_VEL
LIN {X 0,Y 329.501,Z 387.853,A -85,B 0,C 180,E1 -14871.443,E2 -14871.443} C_VEL
LIN {X 0,Y 326.739,Z 374.893,A -85,B 0,C 180,E1 -14872.204,E2 -14872.204} C_VEL
LIN {X 0,Y 326.153,Z 372.08,A -85,B 0,C 180,E1 -14872.377,E2 -14872.377} C_VEL
LIN {X 0,Y 326.691,Z 366.078,A -85,B 0,C 180,E1 -14876.167,E2 -14876.167} C_VEL
LIN {X 0,Y 327.284,Z 360.699,A -85,B 0,C 180,E1 -14879.596,E2 -14879.596} C_VEL
LIN {X 0,Y 327.994,Z 354.988,A -85,B 0,C 180,E1 -14883.315,E2 -14883.315} C_VEL
LIN {X 0,Y 328.288,Z 351.627,A -85,B 0,C 180,E1 -14885.56,E2 -14885.56} C_VEL
LIN {X 0,Y 328.131,Z 347.616,A -85,B 0,C 180,E1 -14888.397,E2 -14888.397} C_VEL
LIN {X 0,Y 327.455,Z 343.265,A -85,B 0,C 180,E1 -14891.707,E2 -14891.707} C_VEL
LIN {X 0,Y 326.666,Z 338.927,A -85,B 0,C 180,E1 -14895.231,E2 -14895.231} C_VEL
LIN {X 0,Y 326.539,Z 338.812,A -85,B 0,C 180,E1 -14898.874,E2 -14898.874} C_VEL
LIN {X 0,Y 326.617,Z 338.802,A -85,B 0,C 180,E1 -14902.762,E2 -14902.762} C_VEL
LIN {X 0,Y 326.6,Z 338.801,A -85,B 0,C 180,E1 -14905.98,E2 -14905.98} C_VEL
LIN {X 0,Y 326.604,Z 338.8,A -85,B 0,C 180,E1 -14909.396,E2 -14909.396} C_VEL
LIN {X 0,Y 326.605,Z 338.8,A -85,B 0,C 180,E1 -14913.135,E2 -14913.135} C_VEL
LIN {X 0,Y 326.625,Z 338.798,A -85,B 0,C 180,E1 -14915.869,E2 -14915.869} C_VEL
LIN {X 0,Y 326.65,Z 338.796,A -85,B 0,C 180,E1 -14919.864,E2 -14919.864} C_VEL
LIN {X 0,Y 326.69,Z 338.791,A -85,B 0,C 180,E1 -14922.472,E2 -14922.472} C_VEL
LIN {X 0,Y 326.75,Z 338.784,A -85,B 0,C 180,E1 -14926.314,E2 -14926.314} C_VEL
LIN {X 0,Y 326.805,Z 338.778,A -85,B 0,C 180,E1 -14930.093,E2 -14930.093} C_VEL
LIN {X 0,Y 326.972,Z 338.754,A -85,B 0,C 180,E1 -14932.59,E2 -14932.59} C_VEL
LIN {X 0,Y 326.773,Z 338.778,A -85,B 0,C 180,E1 -14935.065,E2 -14935.065} C_VEL
LIN {X 0,Y 327.039,Z 338.748,A -85,B 0,C 180,E1 -14937.537,E2 -14937.537} C_VEL
LIN {X 0,Y 327.114,Z 338.738,A -85,B 0,C 180,E1 -14940,E2 -14940} C_VEL
LIN {X 0,Y 327.037,Z 338.745,A -85,B 0,C 180,E1 -14942.463,E2 -14942.463} C_VEL
LIN {X 0,Y 326.964,Z 338.754,A -85,B 0,C 180,E1 -14946.602,E2 -14946.602} C_VEL
LIN {X 0,Y 326.805,Z 338.776,A -85,B 0,C 180,E1 -14949.907,E2 -14949.907} C_VEL
LIN {X 0,Y 326.75,Z 338.783,A -85,B 0,C 180,E1 -14953.686,E2 -14953.686} C_VEL
LIN {X 0,Y 326.691,Z 338.791,A -85,B 0,C 180,E1 -14957.528,E2 -14957.528} C_VEL
LIN {X 0,Y 326.653,Z 338.793,A -85,B 0,C 180,E1 -14960.136,E2 -14960.136} C_VEL
LIN {X 0,Y 326.626,Z 338.796,A -85,B 0,C 180,E1 -14964.131,E2 -14964.131} C_VEL
LIN {X 0,Y 326.591,Z 338.801,A -85,B 0,C 180,E1 -14968.257,E2 -14968.257} C_VEL
LIN {X 0,Y 326.566,Z 338.807,A -85,B 0,C 180,E1 -14971.098,E2 -14971.098} C_VEL
LIN {X 0,Y 326.601,Z 338.8,A -85,B 0,C 180,E1 -14974.02,E2 -14974.02} C_VEL
LIN {X 0,Y 326.617,Z 338.799,A -85,B 0,C 180,E1 -14977.238,E2 -14977.238} C_VEL
LIN {X 0,Y 326.538,Z 338.809,A -85,B 0,C 180,E1 -14981.125,E2 -14981.125} C_VEL
LIN {X 0,Y 326.556,Z 338.805,A -85,B 0,C 180,E1 -14983.527,E2 -14983.527} C_VEL
LIN {X 0,Y 326.595,Z 338.802,A -85,B 0,C 180,E1 -14987.025,E2 -14987.025} C_VEL
LIN {X 0,Y 326.61,Z 338.802,A -85,B 0,C 180,E1 -14990.774,E2 -14990.774} C_VEL
LIN {X 0,Y 326.608,Z 339.24,A -85,B 0,C 180,E1 -14992.952,E2 -14992.952} C_VEL
LIN {X 0,Y 326.602,Z 342.212,A -85,B 0,C 180,E1 -14995.981,E2 -14995.981} C_VEL
LIN {X 0,Y 326.346,Z 345.793,A -85,B 0,C 180,E1 -14999.476,E2 -14999.476} C_VEL
LIN {X 0,Y 326.067,Z 349.662,A -85,B 0,C 180,E1 -15003.089,E2 -15003.089} C_VEL
LIN {X 0,Y 325.859,Z 352.702,A -85,B 0,C 180,E1 -15005.81,E2 -15005.81} C_VEL
LIN {X 0,Y 325.768,Z 354.91,A -85,B 0,C 180,E1 -15007.718,E2 -15007.718} C_VEL
LIN {X 0,Y 329.408,Z 368.003,A -85,B 0,C 180,E1 -15008.532,E2 -15008.532} C_VEL
LIN {X 0,Y 332.087,Z 379.848,A -85,B 0,C 180,E1 -15009.455,E2 -15009.455} C_VEL
LIN {X 0,Y 333.654,Z 389.104,A -85,B 0,C 180,E1 -15010.306,E2 -15010.306} C_VEL
LIN {X 0,Y 332.562,Z 400.189,A -85,B 0,C 180,E1 -15011.36,E2 -15011.36} C_VEL
LIN {X 0,Y 331.322,Z 411.006,A -85,B 0,C 180,E1 -15012.658,E2 -15012.658} C_VEL
LIN {X 0,Y 330.271,Z 419.642,A -85,B 0,C 180,E1 -15013.942,E2 -15013.942} C_VEL
LIN {X 0,Y 329.023,Z 428.13,A -85,B 0,C 180,E1 -15015.465,E2 -15015.465} C_VEL
LIN {X 0,Y 327.86,Z 436.375,A -85,B 0,C 180,E1 -15017.308,E2 -15017.308} C_VEL
LIN {X 0,Y 326.995,Z 442.016,A -85,B 0,C 180,E1 -15018.848,E2 -15018.848} C_VEL
LIN {X 0,Y 326.172,Z 447.513,A -85,B 0,C 180,E1 -15020.701,E2 -15020.701} C_VEL
LIN {X 0,Y 325.624,Z 451.825,A -85,B 0,C 180,E1 -15022.56,E2 -15022.56} C_VEL
LIN {X 0,Y 325.429,Z 454.104,A -85,B 0,C 180,E1 -15023.802,E2 -15023.802} C_VEL
LIN {X 0,Y 325.237,Z 455.959,A -85,B 0,C 180,E1 -15025.042,E2 -15025.042} C_VEL
LIN {X 0,Y 325.059,Z 457.356,A -85,B 0,C 180,E1 -15026.282,E2 -15026.282} C_VEL
LIN {X 0,Y 324.889,Z 458.96,A -85,B 0,C 180,E1 -15028.761,E2 -15028.761} C_VEL
LIN {X 0,Y 324.883,Z 459.19,A -85,B 0,C 180,E1 -15030.001,E2 -15030.001} C_VEL
LIN {X 0,Y 324.889,Z 458.999,A -85,B 0,C 180,E1 -15031.24,E2 -15031.24} C_VEL
LIN {X 0,Y 325.058,Z 457.446,A -85,B 0,C 180,E1 -15033.719,E2 -15033.719} C_VEL
LIN {X 0,Y 325.234,Z 456.089,A -85,B 0,C 180,E1 -15034.959,E2 -15034.959} C_VEL
LIN {X 0,Y 325.551,Z 453.329,A -85,B 0,C 180,E1 -15036.757,E2 -15036.757} C_VEL
LIN {X 0,Y 325.914,Z 449.341,A -85,B 0,C 180,E1 -15038.682,E2 -15038.682} C_VEL
LIN {X 0,Y 326.68,Z 444.324,A -85,B 0,C 180,E1 -15040.537,E2 -15040.537} C_VEL
LIN {X 0,Y 327.593,Z 438.009,A -85,B 0,C 180,E1 -15042.389,E2 -15042.389} C_VEL
LIN {X 0,Y 328.731,Z 430.103,A -85,B 0,C 180,E1 -15044.233,E2 -15044.233} C_VEL
LIN {X 0,Y 330.211,Z 420.264,A -85,B 0,C 180,E1 -15046.063,E2 -15046.063} C_VEL
LIN {X 0,Y 331.439,Z 409.939,A -85,B 0,C 180,E1 -15047.588,E2 -15047.588} C_VEL
LIN {X 0,Y 332.644,Z 399.707,A -85,B 0,C 180,E1 -15048.796,E2 -15048.796} C_VEL
LIN {X 0,Y 333.658,Z 390.268,A -85,B 0,C 180,E1 -15049.695,E2 -15049.695} C_VEL
LIN {X 0,Y 332.235,Z 380.792,A -85,B 0,C 180,E1 -15050.576,E2 -15050.576} C_VEL
LIN {X 0,Y 329.325,Z 367.475,A -85,B 0,C 180,E1 -15051.611,E2 -15051.611} C_VEL
LIN {X 0,Y 325.756,Z 354.869,A -85,B 0,C 180,E1 -15052.406,E2 -15052.406} C_VEL
LIN {X 0,Y 325.949,Z 351.293,A -85,B 0,C 180,E1 -15055.546,E2 -15055.546} C_VEL
LIN {X 0,Y 326.172,Z 348.304,A -85,B 0,C 180,E1 -15058.296,E2 -15058.296} C_VEL
LIN {X 0,Y 326.383,Z 345.306,A -85,B 0,C 180,E1 -15061.117,E2 -15061.117} C_VEL
LIN {X 0,Y 326.606,Z 342.324,A -85,B 0,C 180,E1 -15064.019,E2 -15064.019} C_VEL
LIN {X 0,Y 326.61,Z 339.187,A -85,B 0,C 180,E1 -15067.234,E2 -15067.234} C_VEL
LIN {X 0,Y 326.608,Z 338.803,A -85,B 0,C 180,E1 -15069.226,E2 -15069.226} C_VEL
LIN {X 0,Y 326.576,Z 338.805,A -85,B 0,C 180,E1 -15072.971,E2 -15072.971} C_VEL
LIN {X 0,Y 326.571,Z 338.806,A -85,B 0,C 180,E1 -15077.029,E2 -15077.029} C_VEL
LIN {X 0,Y 326.581,Z 338.807,A -85,B 0,C 180,E1 -15081.385,E2 -15081.385} C_VEL
LIN {X 0,Y 326.618,Z 338.799,A -85,B 0,C 180,E1 -15084.851,E2 -15084.851} C_VEL
LIN {X 0,Y 326.606,Z 338.802,A -85,B 0,C 180,E1 -15087.455,E2 -15087.455} C_VEL
LIN {X 0,Y 326.561,Z 338.805,A -85,B 0,C 180,E1 -15088.614,E2 -15088.614} C_VEL
LIN {X 0,Y 325.913,Z 338.89,A -85,B 0,C 180,E1 -15089.644,E2 -15089.644} C_VEL
LIN {X 0,Y 323.066,Z 339.244,A -85,B 0,C 180,E1 -15091.32,E2 -15091.32} C_VEL
LIN {X 0,Y 320.656,Z 339.542,A -85,B 0,C 180,E1 -15092.678,E2 -15092.678} C_VEL
LIN {X 0,Y 319.643,Z 339.667,A -85,B 0,C 180,E1 -15093.729,E2 -15093.729} C_VEL
LIN {X 0,Y 319.572,Z 339.675,A -85,B 0,C 180,E1 -15094.085,E2 -15094.085} C_VEL
LIN {X 0,Y 319.565,Z 339.676,A -85,B 0,C 180,E1 -15098.045,E2 -15098.045} C_VEL
LIN {X 0,Y 319.687,Z 339.665,A -85,B 0,C 180,E1 -15100.962,E2 -15100.962} C_VEL
LIN {X 0,Y 319.729,Z 339.657,A -85,B 0,C 180,E1 -15105.276,E2 -15105.276} C_VEL
LIN {X 0,Y 319.755,Z 339.653,A -85,B 0,C 180,E1 -15109.873,E2 -15109.873} C_VEL
LIN {X 0,Y 319.932,Z 339.635,A -85,B 0,C 180,E1 -15112.426,E2 -15112.426} C_VEL
LIN {X 0,Y 319.744,Z 339.655,A -85,B 0,C 180,E1 -15114.956,E2 -15114.956} C_VEL
LIN {X 0,Y 319.986,Z 339.623,A -85,B 0,C 180,E1 -15117.482,E2 -15117.482} C_VEL
LIN {X 0,Y 320.075,Z 339.615,A -85,B 0,C 180,E1 -15120,E2 -15120} C_VEL
LIN {X 0,Y 319.986,Z 339.627,A -85,B 0,C 180,E1 -15122.518,E2 -15122.518} C_VEL
LIN {X 0,Y 319.941,Z 339.634,A -85,B 0,C 180,E1 -15126.306,E2 -15126.306} C_VEL
LIN {X 0,Y 319.835,Z 339.643,A -85,B 0,C 180,E1 -15128.848,E2 -15128.848} C_VEL
LIN {X 0,Y 319.679,Z 339.663,A -85,B 0,C 180,E1 -15132.7,E2 -15132.7} C_VEL
LIN {X 0,Y 319.697,Z 339.661,A -85,B 0,C 180,E1 -15135.296,E2 -15135.296} C_VEL
LIN {X 0,Y 319.671,Z 339.664,A -85,B 0,C 180,E1 -15139.255,E2 -15139.255} C_VEL
LIN {X 0,Y 319.551,Z 339.68,A -85,B 0,C 180,E1 -15143.321,E2 -15143.321} C_VEL
LIN {X 0,Y 319.568,Z 339.678,A -85,B 0,C 180,E1 -15146.094,E2 -15146.094} C_VEL
LIN {X 0,Y 319.54,Z 339.681,A -85,B 0,C 180,E1 -15148.939,E2 -15148.939} C_VEL
LIN {X 0,Y 319.522,Z 339.685,A -85,B 0,C 180,E1 -15151.863,E2 -15151.863} C_VEL
LIN {X 0,Y 319.578,Z 339.679,A -85,B 0,C 180,E1 -15155.543,E2 -15155.543} C_VEL
LIN {X 0,Y 319.527,Z 339.683,A -85,B 0,C 180,E1 -15159.662,E2 -15159.662} C_VEL
LIN {X 0,Y 319.517,Z 339.685,A -85,B 0,C 180,E1 -15163.46,E2 -15163.46} C_VEL
LIN {X 0,Y 319.539,Z 339.904,A -85,B 0,C 180,E1 -15164.386,E2 -15164.386} C_VEL
LIN {X 0,Y 320.404,Z 344.477,A -85,B 0,C 180,E1 -15168.227,E2 -15168.227} C_VEL
LIN {X 0,Y 320.894,Z 347.5,A -85,B 0,C 180,E1 -15170.57,E2 -15170.57} C_VEL
LIN {X 0,Y 321.229,Z 350.765,A -85,B 0,C 180,E1 -15173.011,E2 -15173.011} C_VEL
LIN {X 0,Y 321.184,Z 354.033,A -85,B 0,C 180,E1 -15175.325,E2 -15175.325} C_VEL
LIN {X 0,Y 320.56,Z 359.112,A -85,B 0,C 180,E1 -15178.765,E2 -15178.765} C_VEL
LIN {X 0,Y 319.866,Z 364.815,A -85,B 0,C 180,E1 -15182.522,E2 -15182.522} C_VEL
LIN {X 0,Y 319.189,Z 371.182,A -85,B 0,C 180,E1 -15186.651,E2 -15186.651} C_VEL
LIN {X 0,Y 319.143,Z 372.044,A -85,B 0,C 180,E1 -15187.14,E2 -15187.14} C_VEL
LIN {X 0,Y 322.09,Z 385.096,A -85,B 0,C 180,E1 -15187.886,E2 -15187.886} C_VEL
LIN {X 0,Y 324.166,Z 397.4,A -85,B 0,C 180,E1 -15188.789,E2 -15188.789} C_VEL
LIN {X 0,Y 325.412,Z 408.546,A -85,B 0,C 180,E1 -15189.784,E2 -15189.784} C_VEL
LIN {X 0,Y 325.698,Z 415.199,A -85,B 0,C 180,E1 -15190.46,E2 -15190.46} C_VEL
LIN {X 0,Y 324.315,Z 426.174,A -85,B 0,C 180,E1 -15191.686,E2 -15191.686} C_VEL
LIN {X 0,Y 322.926,Z 436.522,A -85,B 0,C 180,E1 -15193.15,E2 -15193.15} C_VEL
LIN {X 0,Y 321.565,Z 445.905,A -85,B 0,C 180,E1 -15194.795,E2 -15194.795} C_VEL
LIN {X 0,Y 320.507,Z 453.211,A -85,B 0,C 180,E1 -15196.365,E2 -15196.365} C_VEL
LIN {X 0,Y 319.465,Z 460.407,A -85,B 0,C 180,E1 -15198.258,E2 -15198.258} C_VEL
LIN {X 0,Y 318.646,Z 466.966,A -85,B 0,C 180,E1 -15200.478,E2 -15200.478} C_VEL
LIN {X 0,Y 318.18,Z 471.307,A -85,B 0,C 180,E1 -15202.384,E2 -15202.384} C_VEL
LIN {X 0,Y 317.902,Z 474.416,A -85,B 0,C 180,E1 -15204.175,E2 -15204.175} C_VEL
LIN {X 0,Y 317.82,Z 476.871,A -85,B 0,C 180,E1 -15206.196,E2 -15206.196} C_VEL
LIN {X 0,Y 317.759,Z 477.869,A -85,B 0,C 180,E1 -15207.464,E2 -15207.464} C_VEL
LIN {X 0,Y 317.727,Z 478.478,A -85,B 0,C 180,E1 -15208.732,E2 -15208.732} C_VEL
LIN {X 0,Y 317.745,Z 478.694,A -85,B 0,C 180,E1 -15209.999,E2 -15209.999} C_VEL
LIN {X 0,Y 317.727,Z 478.475,A -85,B 0,C 180,E1 -15211.267,E2 -15211.267} C_VEL
LIN {X 0,Y 317.759,Z 477.865,A -85,B 0,C 180,E1 -15212.535,E2 -15212.535} C_VEL
LIN {X 0,Y 317.819,Z 476.867,A -85,B 0,C 180,E1 -15213.803,E2 -15213.803} C_VEL
LIN {X 0,Y 317.9,Z 474.412,A -85,B 0,C 180,E1 -15215.82,E2 -15215.82} C_VEL
LIN {X 0,Y 318.15,Z 471.289,A -85,B 0,C 180,E1 -15217.616,E2 -15217.616} C_VEL
LIN {X 0,Y 318.647,Z 466.941,A -85,B 0,C 180,E1 -15219.521,E2 -15219.521} C_VEL
LIN {X 0,Y 319.327,Z 461.403,A -85,B 0,C 180,E1 -15221.424,E2 -15221.424} C_VEL
LIN {X 0,Y 320.331,Z 454.495,A -85,B 0,C 180,E1 -15223.318,E2 -15223.318} C_VEL
LIN {X 0,Y 321.395,Z 447.445,A -85,B 0,C 180,E1 -15224.888,E2 -15224.888} C_VEL
LIN {X 0,Y 322.648,Z 438.161,A -85,B 0,C 180,E1 -15226.58,E2 -15226.58} C_VEL
LIN {X 0,Y 324.073,Z 427.273,A -85,B 0,C 180,E1 -15228.163,E2 -15228.163} C_VEL
LIN {X 0,Y 325.528,Z 416.643,A -85,B 0,C 180,E1 -15229.386,E2 -15229.386} C_VEL
LIN {X 0,Y 325.719,Z 411.917,A -85,B 0,C 180,E1 -15229.866,E2 -15229.866} C_VEL
LIN {X 0,Y 324.474,Z 399.857,A -85,B 0,C 180,E1 -15230.997,E2 -15230.997} C_VEL
LIN {X 0,Y 322.459,Z 387.076,A -85,B 0,C 180,E1 -15231.965,E2 -15231.965} C_VEL
LIN {X 0,Y 319.639,Z 374.34,A -85,B 0,C 180,E1 -15232.736,E2 -15232.736} C_VEL
LIN {X 0,Y 319.157,Z 371.9,A -85,B 0,C 180,E1 -15232.873,E2 -15232.873} C_VEL
LIN {X 0,Y 319.738,Z 365.872,A -85,B 0,C 180,E1 -15236.781,E2 -15236.781} C_VEL
LIN {X 0,Y 320.342,Z 360.504,A -85,B 0,C 180,E1 -15240.303,E2 -15240.303} C_VEL
LIN {X 0,Y 321.036,Z 355.422,A -85,B 0,C 180,E1 -15243.707,E2 -15243.707} C_VEL
LIN {X 0,Y 321.243,Z 351.815,A -85,B 0,C 180,E1 -15246.205,E2 -15246.205} C_VEL
LIN {X 0,Y 320.959,Z 347.435,A -85,B 0,C 180,E1 -15249.419,E2 -15249.419} C_VEL
LIN {X 0,Y 320.248,Z 343.099,A -85,B 0,C 180,E1 -15252.866,E2 -15252.866} C_VEL
LIN {X 0,Y 319.571,Z 339.68,A -85,B 0,C 180,E1 -15255.79,E2 -15255.79} C_VEL
LIN {X 0,Y 319.494,Z 339.689,A -85,B 0,C 180,E1 -15258.706,E2 -15258.706} C_VEL
LIN {X 0,Y 319.54,Z 339.683,A -85,B 0,C 180,E1 -15262.35,E2 -15262.35} C_VEL
LIN {X 0,Y 319.553,Z 339.68,A -85,B 0,C 180,E1 -15265.122,E2 -15265.122} C_VEL
LIN {X 0,Y 319.517,Z 339.685,A -85,B 0,C 180,E1 -15268.136,E2 -15268.136} C_VEL
LIN {X 0,Y 319.563,Z 339.677,A -85,B 0,C 180,E1 -15271.603,E2 -15271.603} C_VEL
LIN {X 0,Y 319.566,Z 339.676,A -85,B 0,C 180,E1 -15275.301,E2 -15275.301} C_VEL
LIN {X 0,Y 319.594,Z 339.673,A -85,B 0,C 180,E1 -15279.4,E2 -15279.4} C_VEL
LIN {X 0,Y 319.65,Z 339.67,A -85,B 0,C 180,E1 -15282.073,E2 -15282.073} C_VEL
LIN {X 0,Y 319.724,Z 339.661,A -85,B 0,C 180,E1 -15286.007,E2 -15286.007} C_VEL
LIN {X 0,Y 319.749,Z 339.657,A -85,B 0,C 180,E1 -15289.873,E2 -15289.873} C_VEL
LIN {X 0,Y 319.926,Z 339.632,A -85,B 0,C 180,E1 -15292.426,E2 -15292.426} C_VEL
LIN {X 0,Y 319.743,Z 339.654,A -85,B 0,C 180,E1 -15294.956,E2 -15294.956} C_VEL
LIN {X 0,Y 319.983,Z 339.626,A -85,B 0,C 180,E1 -15297.482,E2 -15297.482} C_VEL
LIN {X 0,Y 320.071,Z 339.616,A -85,B 0,C 180,E1 -15300,E2 -15300} C_VEL
LIN {X 0,Y 319.981,Z 339.623,A -85,B 0,C 180,E1 -15302.518,E2 -15302.518} C_VEL
LIN {X 0,Y 319.926,Z 339.63,A -85,B 0,C 180,E1 -15306.592,E2 -15306.592} C_VEL
LIN {X 0,Y 319.834,Z 339.642,A -85,B 0,C 180,E1 -15308.848,E2 -15308.848} C_VEL
LIN {X 0,Y 319.673,Z 339.663,A -85,B 0,C 180,E1 -15312.7,E2 -15312.7} C_VEL
LIN {X 0,Y 319.691,Z 339.665,A -85,B 0,C 180,E1 -15315.296,E2 -15315.296} C_VEL
LIN {X 0,Y 319.666,Z 339.668,A -85,B 0,C 180,E1 -15319.256,E2 -15319.256} C_VEL
LIN {X 0,Y 319.554,Z 339.68,A -85,B 0,C 180,E1 -15323.321,E2 -15323.321} C_VEL
LIN {X 0,Y 319.562,Z 339.676,A -85,B 0,C 180,E1 -15326.095,E2 -15326.095} C_VEL
LIN {X 0,Y 319.535,Z 339.684,A -85,B 0,C 180,E1 -15328.939,E2 -15328.939} C_VEL
LIN {X 0,Y 319.517,Z 339.682,A -85,B 0,C 180,E1 -15331.864,E2 -15331.864} C_VEL
LIN {X 0,Y 319.573,Z 339.675,A -85,B 0,C 180,E1 -15335.544,E2 -15335.544} C_VEL
LIN {X 0,Y 319.522,Z 339.682,A -85,B 0,C 180,E1 -15339.663,E2 -15339.663} C_VEL
LIN {X 0,Y 319.515,Z 339.682,A -85,B 0,C 180,E1 -15343.461,E2 -15343.461} C_VEL
LIN {X 0,Y 319.571,Z 339.677,A -85,B 0,C 180,E1 -15347.021,E2 -15347.021} C_VEL
LIN {X 0,Y 319.548,Z 339.683,A -85,B 0,C 180,E1 -15350.373,E2 -15350.373} C_VEL
LIN {X 0,Y 319.535,Z 339.779,A -85,B 0,C 180,E1 -15352.355,E2 -15352.355} C_VEL
LIN {X 0,Y 319.62,Z 342.389,A -85,B 0,C 180,E1 -15355.132,E2 -15355.132} C_VEL
LIN {X 0,Y 319.409,Z 345.368,A -85,B 0,C 180,E1 -15358.126,E2 -15358.126} C_VEL
LIN {X 0,Y 319.193,Z 349.097,A -85,B 0,C 180,E1 -15361.73,E2 -15361.73} C_VEL
LIN {X 0,Y 318.862,Z 352.91,A -85,B 0,C 180,E1 -15365.244,E2 -15365.244} C_VEL
LIN {X 0,Y 318.728,Z 355.097,A -85,B 0,C 180,E1 -15367.195,E2 -15367.195} C_VEL
LIN {X 0,Y 322.482,Z 368.289,A -85,B 0,C 180,E1 -15368.05,E2 -15368.05} C_VEL
LIN {X 0,Y 325.169,Z 380.081,A -85,B 0,C 180,E1 -15368.997,E2 -15368.997} C_VEL
LIN {X 0,Y 326.91,Z 391.085,A -85,B 0,C 180,E1 -15370.046,E2 -15370.046} C_VEL
LIN {X 0,Y 325.698,Z 401.83,A -85,B 0,C 180,E1 -15371.116,E2 -15371.116} C_VEL
LIN {X 0,Y 324.508,Z 411.705,A -85,B 0,C 180,E1 -15372.351,E2 -15372.351} C_VEL
LIN {X 0,Y 323.458,Z 419.861,A -85,B 0,C 180,E1 -15373.594,E2 -15373.594} C_VEL
LIN {X 0,Y 322.163,Z 428.348,A -85,B 0,C 180,E1 -15375.149,E2 -15375.149} C_VEL
LIN {X 0,Y 320.917,Z 436.593,A -85,B 0,C 180,E1 -15377.029,E2 -15377.029} C_VEL
LIN {X 0,Y 320.03,Z 442.233,A -85,B 0,C 180,E1 -15378.602,E2 -15378.602} C_VEL
LIN {X 0,Y 319.172,Z 447.73,A -85,B 0,C 180,E1 -15380.495,E2 -15380.495} C_VEL
LIN {X 0,Y 318.584,Z 452.042,A -85,B 0,C 180,E1 -15382.395,E2 -15382.395} C_VEL
LIN {X 0,Y 318.384,Z 454.32,A -85,B 0,C 180,E1 -15383.664,E2 -15383.664} C_VEL
LIN {X 0,Y 318.167,Z 456.175,A -85,B 0,C 180,E1 -15384.932,E2 -15384.932} C_VEL
LIN {X 0,Y 317.994,Z 457.571,A -85,B 0,C 180,E1 -15386.199,E2 -15386.199} C_VEL
LIN {X 0,Y 317.8,Z 459.175,A -85,B 0,C 180,E1 -15388.733,E2 -15388.733} C_VEL
LIN {X 0,Y 317.79,Z 459.406,A -85,B 0,C 180,E1 -15390.001,E2 -15390.001} C_VEL
LIN {X 0,Y 317.799,Z 459.214,A -85,B 0,C 180,E1 -15391.268,E2 -15391.268} C_VEL
LIN {X 0,Y 317.993,Z 457.661,A -85,B 0,C 180,E1 -15393.802,E2 -15393.802} C_VEL
LIN {X 0,Y 318.164,Z 456.304,A -85,B 0,C 180,E1 -15395.07,E2 -15395.07} C_VEL
LIN {X 0,Y 318.469,Z 453.807,A -85,B 0,C 180,E1 -15396.749,E2 -15396.749} C_VEL
LIN {X 0,Y 318.899,Z 449.556,A -85,B 0,C 180,E1 -15398.875,E2 -15398.875} C_VEL
LIN {X 0,Y 319.704,Z 444.538,A -85,B 0,C 180,E1 -15400.77,E2 -15400.77} C_VEL
LIN {X 0,Y 320.661,Z 438.222,A -85,B 0,C 180,E1 -15402.661,E2 -15402.661} C_VEL
LIN {X 0,Y 321.856,Z 430.316,A -85,B 0,C 180,E1 -15404.544,E2 -15404.544} C_VEL
LIN {X 0,Y 323.393,Z 420.476,A -85,B 0,C 180,E1 -15406.411,E2 -15406.411} C_VEL
LIN {X 0,Y 324.663,Z 410.151,A -85,B 0,C 180,E1 -15407.967,E2 -15407.967} C_VEL
LIN {X 0,Y 326.091,Z 398.496,A -85,B 0,C 180,E1 -15409.352,E2 -15409.352} C_VEL
LIN {X 0,Y 326.901,Z 390.479,A -85,B 0,C 180,E1 -15410.12,E2 -15410.12} C_VEL
LIN {X 0,Y 324.991,Z 379.27,A -85,B 0,C 180,E1 -15411.185,E2 -15411.185} C_VEL
LIN {X 0,Y 322.024,Z 366.614,A -85,B 0,C 180,E1 -15412.186,E2 -15412.186} C_VEL
LIN {X 0,Y 318.726,Z 355.081,A -85,B 0,C 180,E1 -15412.932,E2 -15412.932} C_VEL
LIN {X 0,Y 318.949,Z 351.501,A -85,B 0,C 180,E1 -15416.148,E2 -15416.148} C_VEL
LIN {X 0,Y 319.173,Z 348.5,A -85,B 0,C 180,E1 -15418.975,E2 -15418.975} C_VEL
LIN {X 0,Y 319.413,Z 345.494,A -85,B 0,C 180,E1 -15421.875,E2 -15421.875} C_VEL
LIN {X 0,Y 319.61,Z 342.496,A -85,B 0,C 180,E1 -15424.87,E2 -15424.87} C_VEL
LIN {X 0,Y 319.529,Z 339.685,A -85,B 0,C 180,E1 -15428.014,E2 -15428.014} C_VEL
LIN {X 0,Y 319.526,Z 339.687,A -85,B 0,C 180,E1 -15431.597,E2 -15431.597} C_VEL
LIN {X 0,Y 319.486,Z 339.69,A -85,B 0,C 180,E1 -15435.256,E2 -15435.256} C_VEL
LIN {X 0,Y 319.502,Z 339.684,A -85,B 0,C 180,E1 -15438.407,E2 -15438.407} C_VEL
LIN {X 0,Y 319.545,Z 339.678,A -85,B 0,C 180,E1 -15442.351,E2 -15442.351} C_VEL
LIN {X 0,Y 319.559,Z 339.681,A -85,B 0,C 180,E1 -15445.123,E2 -15445.123} C_VEL
LIN {X 0,Y 319.525,Z 339.681,A -85,B 0,C 180,E1 -15448.62,E2 -15448.62} C_VEL
LIN {X 0,Y 319.542,Z 339.679,A -85,B 0,C 180,E1 -15452.492,E2 -15452.492} C_VEL
LIN {X 0,Y 319.572,Z 339.675,A -85,B 0,C 180,E1 -15454.085,E2 -15454.085} C_VEL
LIN {X 0,Y 318.927,Z 339.759,A -85,B 0,C 180,E1 -15455.138,E2 -15455.138} C_VEL
LIN {X 0,Y 316.058,Z 340.117,A -85,B 0,C 180,E1 -15456.85,E2 -15456.85} C_VEL
LIN {X 0,Y 313.626,Z 340.418,A -85,B 0,C 180,E1 -15458.238,E2 -15458.238} C_VEL
LIN {X 0,Y 312.608,Z 340.545,A -85,B 0,C 180,E1 -15459.314,E2 -15459.314} C_VEL
LIN {X 0,Y 312.539,Z 340.551,A -85,B 0,C 180,E1 -15459.678,E2 -15459.678} C_VEL
LIN {X 0,Y 312.605,Z 340.547,A -85,B 0,C 180,E1 -15463.006,E2 -15463.006} C_VEL
LIN {X 0,Y 312.691,Z 340.532,A -85,B 0,C 180,E1 -15465.686,E2 -15465.686} C_VEL
LIN {X 0,Y 312.699,Z 340.531,A -85,B 0,C 180,E1 -15469.642,E2 -15469.642} C_VEL
LIN {X 0,Y 312.871,Z 340.513,A -85,B 0,C 180,E1 -15472.254,E2 -15472.254} C_VEL
LIN {X 0,Y 312.714,Z 340.531,A -85,B 0,C 180,E1 -15474.842,E2 -15474.842} C_VEL
LIN {X 0,Y 312.933,Z 340.502,A -85,B 0,C 180,E1 -15477.426,E2 -15477.426} C_VEL
LIN {X 0,Y 313.033,Z 340.492,A -85,B 0,C 180,E1 -15480,E2 -15480} C_VEL
LIN {X 0,Y 312.932,Z 340.505,A -85,B 0,C 180,E1 -15482.574,E2 -15482.574} C_VEL
LIN {X 0,Y 312.898,Z 340.51,A -85,B 0,C 180,E1 -15486.448,E2 -15486.448} C_VEL
LIN {X 0,Y 312.765,Z 340.523,A -85,B 0,C 180,E1 -15489.05,E2 -15489.05} C_VEL
LIN {X 0,Y 312.631,Z 340.54,A -85,B 0,C 180,E1 -15492.991,E2 -15492.991} C_VEL
LIN {X 0,Y 312.636,Z 340.543,A -85,B 0,C 180,E1 -15495.65,E2 -15495.65} C_VEL
LIN {X 0,Y 312.627,Z 340.542,A -85,B 0,C 180,E1 -15499.236,E2 -15499.236} C_VEL
LIN {X 0,Y 312.522,Z 340.554,A -85,B 0,C 180,E1 -15502.78,E2 -15502.78} C_VEL
LIN {X 0,Y 312.527,Z 340.556,A -85,B 0,C 180,E1 -15505.908,E2 -15505.908} C_VEL
LIN {X 0,Y 312.493,Z 340.562,A -85,B 0,C 180,E1 -15509.655,E2 -15509.655} C_VEL
LIN {X 0,Y 312.518,Z 340.559,A -85,B 0,C 180,E1 -15513.689,E2 -15513.689} C_VEL
LIN {X 0,Y 312.513,Z 340.559,A -85,B 0,C 180,E1 -15517.387,E2 -15517.387} C_VEL
LIN {X 0,Y 312.439,Z 340.565,A -85,B 0,C 180,E1 -15520.717,E2 -15520.717} C_VEL
LIN {X 0,Y 312.511,Z 340.665,A -85,B 0,C 180,E1 -15523.86,E2 -15523.86} C_VEL
LIN {X 0,Y 313.32,Z 345.188,A -85,B 0,C 180,E1 -15527.75,E2 -15527.75} C_VEL
LIN {X 0,Y 313.982,Z 349.49,A -85,B 0,C 180,E1 -15531.19,E2 -15531.19} C_VEL
LIN {X 0,Y 314.221,Z 352.738,A -85,B 0,C 180,E1 -15533.629,E2 -15533.629} C_VEL
LIN {X 0,Y 314.043,Z 356.028,A -85,B 0,C 180,E1 -15535.98,E2 -15535.98} C_VEL
LIN {X 0,Y 313.465,Z 360.328,A -85,B 0,C 180,E1 -15538.958,E2 -15538.958} C_VEL
LIN {X 0,Y 312.786,Z 365.687,A -85,B 0,C 180,E1 -15542.573,E2 -15542.573} C_VEL
LIN {X 0,Y 312.123,Z 371.683,A -85,B 0,C 180,E1 -15546.573,E2 -15546.573} C_VEL
LIN {X 0,Y 315.378,Z 386.012,A -85,B 0,C 180,E1 -15547.454,E2 -15547.454} C_VEL
LIN {X 0,Y 317.447,Z 398.425,A -85,B 0,C 180,E1 -15548.411,E2 -15548.411} C_VEL
LIN {X 0,Y 318.666,Z 410.107,A -85,B 0,C 180,E1 -15549.506,E2 -15549.506} C_VEL
LIN {X 0,Y 318.955,Z 414.987,A -85,B 0,C 180,E1 -15550.029,E2 -15550.029} C_VEL
LIN {X 0,Y 317.542,Z 425.961,A -85,B 0,C 180,E1 -15551.281,E2 -15551.281} C_VEL
LIN {X 0,Y 316.135,Z 435.967,A -85,B 0,C 180,E1 -15552.719,E2 -15552.719} C_VEL
LIN {X 0,Y 314.701,Z 445.691,A -85,B 0,C 180,E1 -15554.455,E2 -15554.455} C_VEL
LIN {X 0,Y 313.59,Z 452.997,A -85,B 0,C 180,E1 -15556.059,E2 -15556.059} C_VEL
LIN {X 0,Y 312.465,Z 460.192,A -85,B 0,C 180,E1 -15557.991,E2 -15557.991} C_VEL
LIN {X 0,Y 311.825,Z 465.053,A -85,B 0,C 180,E1 -15559.612,E2 -15559.612} C_VEL
LIN {X 0,Y 311.252,Z 469.779,A -85,B 0,C 180,E1 -15561.56,E2 -15561.56} C_VEL
LIN {X 0,Y 310.906,Z 473.392,A -85,B 0,C 180,E1 -15563.51,E2 -15563.51} C_VEL
LIN {X 0,Y 310.769,Z 475.256,A -85,B 0,C 180,E1 -15564.809,E2 -15564.809} C_VEL
LIN {X 0,Y 310.733,Z 476.656,A -85,B 0,C 180,E1 -15566.109,E2 -15566.109} C_VEL
LIN {X 0,Y 310.683,Z 477.655,A -85,B 0,C 180,E1 -15567.406,E2 -15567.406} C_VEL
LIN {X 0,Y 310.643,Z 478.263,A -85,B 0,C 180,E1 -15568.703,E2 -15568.703} C_VEL
LIN {X 0,Y 310.656,Z 478.479,A -85,B 0,C 180,E1 -15569.999,E2 -15569.999} C_VEL
LIN {X 0,Y 310.642,Z 478.26,A -85,B 0,C 180,E1 -15571.296,E2 -15571.296} C_VEL
LIN {X 0,Y 310.683,Z 477.65,A -85,B 0,C 180,E1 -15572.592,E2 -15572.592} C_VEL
LIN {X 0,Y 310.731,Z 476.651,A -85,B 0,C 180,E1 -15573.89,E2 -15573.89} C_VEL
LIN {X 0,Y 310.813,Z 474.435,A -85,B 0,C 180,E1 -15575.78,E2 -15575.78} C_VEL
LIN {X 0,Y 311.079,Z 471.071,A -85,B 0,C 180,E1 -15577.79,E2 -15577.79} C_VEL
LIN {X 0,Y 311.619,Z 466.723,A -85,B 0,C 180,E1 -15579.738,E2 -15579.738} C_VEL
LIN {X 0,Y 312.322,Z 461.184,A -85,B 0,C 180,E1 -15581.684,E2 -15581.684} C_VEL
LIN {X 0,Y 313.403,Z 454.277,A -85,B 0,C 180,E1 -15583.618,E2 -15583.618} C_VEL
LIN {X 0,Y 314.482,Z 447.226,A -85,B 0,C 180,E1 -15585.223,E2 -15585.223} C_VEL
LIN {X 0,Y 315.712,Z 438.728,A -85,B 0,C 180,E1 -15586.821,E2 -15586.821} C_VEL
LIN {X 0,Y 317.147,Z 428.23,A -85,B 0,C 180,E1 -15588.407,E2 -15588.407} C_VEL
LIN {X 0,Y 318.814,Z 416.423,A -85,B 0,C 180,E1 -15589.811,E2 -15589.811} C_VEL
LIN {X 0,Y 318.67,Z 409.981,A -85,B 0,C 180,E1 -15590.493,E2 -15590.493} C_VEL
LIN {X 0,Y 317.415,Z 398.453,A -85,B 0,C 180,E1 -15591.575,E2 -15591.575} C_VEL
LIN {X 0,Y 315.251,Z 385.432,A -85,B 0,C 180,E1 -15592.573,E2 -15592.573} C_VEL
LIN {X 0,Y 312.299,Z 372.846,A -85,B 0,C 180,E1 -15593.345,E2 -15593.345} C_VEL
LIN {X 0,Y 312.171,Z 371.667,A -85,B 0,C 180,E1 -15593.419,E2 -15593.419} C_VEL
LIN {X 0,Y 312.783,Z 365.665,A -85,B 0,C 180,E1 -15597.426,E2 -15597.426} C_VEL
LIN {X 0,Y 313.459,Z 360.309,A -85,B 0,C 180,E1 -15601.041,E2 -15601.041} C_VEL
LIN {X 0,Y 314.07,Z 355.867,A -85,B 0,C 180,E1 -15604.111,E2 -15604.111} C_VEL
LIN {X 0,Y 314.206,Z 351.635,A -85,B 0,C 180,E1 -15607.15,E2 -15607.15} C_VEL
LIN {X 0,Y 313.735,Z 347.284,A -85,B 0,C 180,E1 -15610.512,E2 -15610.512} C_VEL
LIN {X 0,Y 313.022,Z 342.953,A -85,B 0,C 180,E1 -15614.106,E2 -15614.106} C_VEL
LIN {X 0,Y 312.523,Z 340.557,A -85,B 0,C 180,E1 -15616.266,E2 -15616.266} C_VEL
LIN {X 0,Y 312.488,Z 340.563,A -85,B 0,C 180,E1 -15620.969,E2 -15620.969} C_VEL
LIN {X 0,Y 312.525,Z 340.556,A -85,B 0,C 180,E1 -15624.219,E2 -15624.219} C_VEL
LIN {X 0,Y 312.494,Z 340.558,A -85,B 0,C 180,E1 -15627.333,E2 -15627.333} C_VEL
LIN {X 0,Y 312.498,Z 340.557,A -85,B 0,C 180,E1 -15631.291,E2 -15631.291} C_VEL
LIN {X 0,Y 312.539,Z 340.554,A -85,B 0,C 180,E1 -15634.707,E2 -15634.707} C_VEL
LIN {X 0,Y 312.556,Z 340.55,A -85,B 0,C 180,E1 -15637.527,E2 -15637.527} C_VEL
LIN {X 0,Y 312.63,Z 340.541,A -85,B 0,C 180,E1 -15641.656,E2 -15641.656} C_VEL
LIN {X 0,Y 312.685,Z 340.535,A -85,B 0,C 180,E1 -15645.686,E2 -15645.686} C_VEL
LIN {X 0,Y 312.693,Z 340.534,A -85,B 0,C 180,E1 -15649.642,E2 -15649.642} C_VEL
LIN {X 0,Y 312.864,Z 340.513,A -85,B 0,C 180,E1 -15652.254,E2 -15652.254} C_VEL
LIN {X 0,Y 312.713,Z 340.529,A -85,B 0,C 180,E1 -15654.842,E2 -15654.842} C_VEL
LIN {X 0,Y 312.93,Z 340.504,A -85,B 0,C 180,E1 -15657.426,E2 -15657.426} C_VEL
LIN {X 0,Y 313.029,Z 340.493,A -85,B 0,C 180,E1 -15660,E2 -15660} C_VEL
LIN {X 0,Y 312.928,Z 340.502,A -85,B 0,C 180,E1 -15662.575,E2 -15662.575} C_VEL
LIN {X 0,Y 312.892,Z 340.507,A -85,B 0,C 180,E1 -15666.574,E2 -15666.574} C_VEL
LIN {X 0,Y 312.779,Z 340.522,A -85,B 0,C 180,E1 -15669.05,E2 -15669.05} C_VEL
LIN {X 0,Y 312.626,Z 340.543,A -85,B 0,C 180,E1 -15672.992,E2 -15672.992} C_VEL
LIN {X 0,Y 312.63,Z 340.542,A -85,B 0,C 180,E1 -15675.65,E2 -15675.65} C_VEL
LIN {X 0,Y 312.622,Z 340.545,A -85,B 0,C 180,E1 -15679.237,E2 -15679.237} C_VEL
LIN {X 0,Y 312.532,Z 340.554,A -85,B 0,C 180,E1 -15682.787,E2 -15682.787} C_VEL
LIN {X 0,Y 312.522,Z 340.553,A -85,B 0,C 180,E1 -15685.909,E2 -15685.909} C_VEL
LIN {X 0,Y 312.488,Z 340.558,A -85,B 0,C 180,E1 -15689.656,E2 -15689.656} C_VEL
LIN {X 0,Y 312.513,Z 340.555,A -85,B 0,C 180,E1 -15693.69,E2 -15693.69} C_VEL
LIN {X 0,Y 312.508,Z 340.556,A -85,B 0,C 180,E1 -15697.388,E2 -15697.388} C_VEL
LIN {X 0,Y 312.435,Z 340.568,A -85,B 0,C 180,E1 -15700.718,E2 -15700.718} C_VEL
LIN {X 0,Y 312.448,Z 340.565,A -85,B 0,C 180,E1 -15704.211,E2 -15704.211} C_VEL
LIN {X 0,Y 312.524,Z 340.556,A -85,B 0,C 180,E1 -15707.911,E2 -15707.911} C_VEL
LIN {X 0,Y 312.479,Z 340.564,A -85,B 0,C 180,E1 -15711.924,E2 -15711.924} C_VEL
LIN {X 0,Y 312.584,Z 342.588,A -85,B 0,C 180,E1 -15714.229,E2 -15714.229} C_VEL
LIN {X 0,Y 312.437,Z 345.56,A -85,B 0,C 180,E1 -15717.327,E2 -15717.327} C_VEL
LIN {X 0,Y 312.14,Z 350.072,A -85,B 0,C 180,E1 -15721.783,E2 -15721.783} C_VEL
LIN {X 0,Y 311.887,Z 353.124,A -85,B 0,C 180,E1 -15724.651,E2 -15724.651} C_VEL
LIN {X 0,Y 311.728,Z 355.476,A -85,B 0,C 180,E1 -15726.658,E2 -15726.658} C_VEL
LIN {X 0,Y 315.567,Z 368.783,A -85,B 0,C 180,E1 -15727.558,E2 -15727.558} C_VEL
LIN {X 0,Y 318.329,Z 380.726,A -85,B 0,C 180,E1 -15728.555,E2 -15728.555} C_VEL
LIN {X 0,Y 320.1,Z 391.312,A -85,B 0,C 180,E1 -15729.603,E2 -15729.603} C_VEL
LIN {X 0,Y 319,Z 402.05,A -85,B 0,C 180,E1 -15730.704,E2 -15730.704} C_VEL
LIN {X 0,Y 317.652,Z 412.581,A -85,B 0,C 180,E1 -15732.059,E2 -15732.059} C_VEL
LIN {X 0,Y 316.378,Z 421.886,A -85,B 0,C 180,E1 -15733.548,E2 -15733.548} C_VEL
LIN {X 0,Y 314.831,Z 431.523,A -85,B 0,C 180,E1 -15735.456,E2 -15735.456} C_VEL
LIN {X 0,Y 313.59,Z 439.205,A -85,B 0,C 180,E1 -15737.379,E2 -15737.379} C_VEL
LIN {X 0,Y 312.45,Z 446.255,A -85,B 0,C 180,E1 -15739.634,E2 -15739.634} C_VEL
LIN {X 0,Y 311.718,Z 450.949,A -85,B 0,C 180,E1 -15741.574,E2 -15741.574} C_VEL
LIN {X 0,Y 311.311,Z 454.537,A -85,B 0,C 180,E1 -15743.519,E2 -15743.519} C_VEL
LIN {X 0,Y 311.101,Z 456.392,A -85,B 0,C 180,E1 -15744.816,E2 -15744.816} C_VEL
LIN {X 0,Y 310.931,Z 457.787,A -85,B 0,C 180,E1 -15746.112,E2 -15746.112} C_VEL
LIN {X 0,Y 310.712,Z 459.39,A -85,B 0,C 180,E1 -15748.705,E2 -15748.705} C_VEL
LIN {X 0,Y 310.701,Z 459.621,A -85,B 0,C 180,E1 -15750.001,E2 -15750.001} C_VEL
LIN {X 0,Y 310.712,Z 459.429,A -85,B 0,C 180,E1 -15751.297,E2 -15751.297} C_VEL
LIN {X 0,Y 310.93,Z 457.875,A -85,B 0,C 180,E1 -15753.889,E2 -15753.889} C_VEL
LIN {X 0,Y 311.099,Z 456.519,A -85,B 0,C 180,E1 -15755.185,E2 -15755.185} C_VEL
LIN {X 0,Y 311.364,Z 454.343,A -85,B 0,C 180,E1 -15756.706,E2 -15756.706} C_VEL
LIN {X 0,Y 311.879,Z 449.77,A -85,B 0,C 180,E1 -15759.076,E2 -15759.076} C_VEL
LIN {X 0,Y 312.723,Z 444.752,A -85,B 0,C 180,E1 -15761.013,E2 -15761.013} C_VEL
LIN {X 0,Y 313.732,Z 438.435,A -85,B 0,C 180,E1 -15762.945,E2 -15762.945} C_VEL
LIN {X 0,Y 314.999,Z 430.528,A -85,B 0,C 180,E1 -15764.867,E2 -15764.867} C_VEL
LIN {X 0,Y 316.594,Z 420.688,A -85,B 0,C 180,E1 -15766.773,E2 -15766.773} C_VEL
LIN {X 0,Y 317.922,Z 410.362,A -85,B 0,C 180,E1 -15768.362,E2 -15768.362} C_VEL
LIN {X 0,Y 319.418,Z 398.706,A -85,B 0,C 180,E1 -15769.773,E2 -15769.773} C_VEL
LIN {X 0,Y 320.144,Z 392.446,A -85,B 0,C 180,E1 -15770.396,E2 -15770.396} C_VEL
LIN {X 0,Y 318.377,Z 380.965,A -85,B 0,C 180,E1 -15771.535,E2 -15771.535} C_VEL
LIN {X 0,Y 315.579,Z 368.806,A -85,B 0,C 180,E1 -15772.552,E2 -15772.552} C_VEL
LIN {X 0,Y 311.803,Z 356.054,A -85,B 0,C 180,E1 -15773.429,E2 -15773.429} C_VEL
LIN {X 0,Y 311.707,Z 355.291,A -85,B 0,C 180,E1 -15773.476,E2 -15773.476} C_VEL
LIN {X 0,Y 311.942,Z 351.712,A -85,B 0,C 180,E1 -15776.782,E2 -15776.782} C_VEL
LIN {X 0,Y 312.195,Z 348.702,A -85,B 0,C 180,E1 -15779.687,E2 -15779.687} C_VEL
LIN {X 0,Y 312.526,Z 344.684,A -85,B 0,C 180,E1 -15783.69,E2 -15783.69} C_VEL
LIN {X 0,Y 312.607,Z 342.501,A -85,B 0,C 180,E1 -15785.967,E2 -15785.967} C_VEL
LIN {X 0,Y 312.482,Z 340.579,A -85,B 0,C 180,E1 -15788.077,E2 -15788.077} C_VEL
LIN {X 0,Y 312.49,Z 340.559,A -85,B 0,C 180,E1 -15790.709,E2 -15790.709} C_VEL
LIN {X 0,Y 312.451,Z 340.565,A -85,B 0,C 180,E1 -15794.209,E2 -15794.209} C_VEL
LIN {X 0,Y 312.453,Z 340.564,A -85,B 0,C 180,E1 -15797.925,E2 -15797.925} C_VEL
LIN {X 0,Y 312.482,Z 340.559,A -85,B 0,C 180,E1 -15801.922,E2 -15801.922} C_VEL
LIN {X 0,Y 312.53,Z 340.553,A -85,B 0,C 180,E1 -15804.22,E2 -15804.22} C_VEL
LIN {X 0,Y 312.5,Z 340.559,A -85,B 0,C 180,E1 -15807.333,E2 -15807.333} C_VEL
LIN {X 0,Y 312.504,Z 340.559,A -85,B 0,C 180,E1 -15811.292,E2 -15811.292} C_VEL
LIN {X 0,Y 312.545,Z 340.553,A -85,B 0,C 180,E1 -15814.707,E2 -15814.707} C_VEL
LIN {X 0,Y 312.561,Z 340.549,A -85,B 0,C 180,E1 -15817.527,E2 -15817.527} C_VEL
LIN {X 0,Y 312.539,Z 340.551,A -85,B 0,C 180,E1 -15819.678,E2 -15819.678} C_VEL
LIN {X 0,Y 311.94,Z 340.63,A -85,B 0,C 180,E1 -15820.753,E2 -15820.753} C_VEL
LIN {X 0,Y 309.207,Z 340.969,A -85,B 0,C 180,E1 -15822.506,E2 -15822.506} C_VEL
LIN {X 0,Y 306.828,Z 341.266,A -85,B 0,C 180,E1 -15823.927,E2 -15823.927} C_VEL
LIN {X 0,Y 305.756,Z 341.399,A -85,B 0,C 180,E1 -15825.025,E2 -15825.025} C_VEL
LIN {X 0,Y 305.642,Z 341.411,A -85,B 0,C 180,E1 -15825.397,E2 -15825.397} C_VEL
LIN {X 0,Y 305.636,Z 341.411,A -85,B 0,C 180,E1 -15829.4,E2 -15829.4} C_VEL
LIN {X 0,Y 305.812,Z 341.391,A -85,B 0,C 180,E1 -15832.074,E2 -15832.074} C_VEL
LIN {X 0,Y 305.686,Z 341.408,A -85,B 0,C 180,E1 -15834.723,E2 -15834.723} C_VEL
LIN {X 0,Y 305.946,Z 341.375,A -85,B 0,C 180,E1 -15838.684,E2 -15838.684} C_VEL
LIN {X 0,Y 305.946,Z 341.372,A -85,B 0,C 180,E1 -15841.316,E2 -15841.316} C_VEL
LIN {X 0,Y 305.683,Z 341.406,A -85,B 0,C 180,E1 -15845.277,E2 -15845.277} C_VEL
LIN {X 0,Y 305.795,Z 341.395,A -85,B 0,C 180,E1 -15847.926,E2 -15847.926} C_VEL
LIN {X 0,Y 305.601,Z 341.42,A -85,B 0,C 180,E1 -15851.945,E2 -15851.945} C_VEL
LIN {X 0,Y 305.635,Z 341.412,A -85,B 0,C 180,E1 -15855.035,E2 -15855.035} C_VEL
LIN {X 0,Y 305.573,Z 341.422,A -85,B 0,C 180,E1 -15859.444,E2 -15859.444} C_VEL
LIN {X 0,Y 305.484,Z 341.431,A -85,B 0,C 180,E1 -15863.039,E2 -15863.039} C_VEL
LIN {X 0,Y 305.467,Z 341.434,A -85,B 0,C 180,E1 -15866.197,E2 -15866.197} C_VEL
LIN {X 0,Y 305.446,Z 341.437,A -85,B 0,C 180,E1 -15869.034,E2 -15869.034} C_VEL
LIN {X 0,Y 305.435,Z 341.439,A -85,B 0,C 180,E1 -15871.953,E2 -15871.953} C_VEL
LIN {X 0,Y 305.461,Z 341.438,A -85,B 0,C 180,E1 -15875.114,E2 -15875.114} C_VEL
LIN {X 0,Y 305.432,Z 341.439,A -85,B 0,C 180,E1 -15878.525,E2 -15878.525} C_VEL
LIN {X 0,Y 305.44,Z 341.437,A -85,B 0,C 180,E1 -15882.583,E2 -15882.583} C_VEL
LIN {X 0,Y 305.457,Z 341.488,A -85,B 0,C 180,E1 -15883.351,E2 -15883.351} C_VEL
LIN {X 0,Y 306.252,Z 345.896,A -85,B 0,C 180,E1 -15887.252,E2 -15887.252} C_VEL
LIN {X 0,Y 306.808,Z 349.291,A -85,B 0,C 180,E1 -15890.105,E2 -15890.105} C_VEL
LIN {X 0,Y 307.197,Z 353.665,A -85,B 0,C 180,E1 -15893.5,E2 -15893.5} C_VEL
LIN {X 0,Y 307.084,Z 356.35,A -85,B 0,C 180,E1 -15895.478,E2 -15895.478} C_VEL
LIN {X 0,Y 306.435,Z 361.198,A -85,B 0,C 180,E1 -15898.934,E2 -15898.934} C_VEL
LIN {X 0,Y 305.716,Z 366.545,A -85,B 0,C 180,E1 -15902.627,E2 -15902.627} C_VEL
LIN {X 0,Y 305.16,Z 371.485,A -85,B 0,C 180,E1 -15906.008,E2 -15906.008} C_VEL
LIN {X 0,Y 308.462,Z 385.794,A -85,B 0,C 180,E1 -15906.919,E2 -15906.919} C_VEL
LIN {X 0,Y 310.601,Z 398.485,A -85,B 0,C 180,E1 -15907.931,E2 -15907.931} C_VEL
LIN {X 0,Y 311.814,Z 409.891,A -85,B 0,C 180,E1 -15909.034,E2 -15909.034} C_VEL
LIN {X 0,Y 312.103,Z 416.31,A -85,B 0,C 180,E1 -15909.744,E2 -15909.744} C_VEL
LIN {X 0,Y 310.463,Z 428.103,A -85,B 0,C 180,E1 -15911.181,E2 -15911.181} C_VEL
LIN {X 0,Y 308.934,Z 438.581,A -85,B 0,C 180,E1 -15912.798,E2 -15912.798} C_VEL
LIN {X 0,Y 307.573,Z 447.061,A -85,B 0,C 180,E1 -15914.426,E2 -15914.426} C_VEL
LIN {X 0,Y 306.274,Z 455.341,A -85,B 0,C 180,E1 -15916.396,E2 -15916.396} C_VEL
LIN {X 0,Y 305.204,Z 462.016,A -85,B 0,C 180,E1 -15918.376,E2 -15918.376} C_VEL
LIN {X 0,Y 304.373,Z 468.129,A -85,B 0,C 180,E1 -15920.698,E2 -15920.698} C_VEL
LIN {X 0,Y 303.944,Z 472.104,A -85,B 0,C 180,E1 -15922.693,E2 -15922.693} C_VEL
LIN {X 0,Y 303.686,Z 475.041,A -85,B 0,C 180,E1 -15924.688,E2 -15924.688} C_VEL
LIN {X 0,Y 303.648,Z 476.441,A -85,B 0,C 180,E1 -15926.018,E2 -15926.018} C_VEL
LIN {X 0,Y 303.609,Z 477.44,A -85,B 0,C 180,E1 -15927.346,E2 -15927.346} C_VEL
LIN {X 0,Y 303.56,Z 478.048,A -85,B 0,C 180,E1 -15928.673,E2 -15928.673} C_VEL
LIN {X 0,Y 303.571,Z 478.264,A -85,B 0,C 180,E1 -15929.999,E2 -15929.999} C_VEL
LIN {X 0,Y 303.56,Z 478.045,A -85,B 0,C 180,E1 -15931.326,E2 -15931.326} C_VEL
LIN {X 0,Y 303.608,Z 477.435,A -85,B 0,C 180,E1 -15932.653,E2 -15932.653} C_VEL
LIN {X 0,Y 303.647,Z 476.435,A -85,B 0,C 180,E1 -15933.981,E2 -15933.981} C_VEL
LIN {X 0,Y 303.729,Z 474.452,A -85,B 0,C 180,E1 -15935.743,E2 -15935.743} C_VEL
LIN {X 0,Y 304.033,Z 470.854,A -85,B 0,C 180,E1 -15937.972,E2 -15937.972} C_VEL
LIN {X 0,Y 304.578,Z 466.505,A -85,B 0,C 180,E1 -15939.965,E2 -15939.965} C_VEL
LIN {X 0,Y 305.322,Z 460.966,A -85,B 0,C 180,E1 -15941.955,E2 -15941.955} C_VEL
LIN {X 0,Y 306.46,Z 454.059,A -85,B 0,C 180,E1 -15943.933,E2 -15943.933} C_VEL
LIN {X 0,Y 307.594,Z 447.007,A -85,B 0,C 180,E1 -15945.572,E2 -15945.572} C_VEL
LIN {X 0,Y 308.901,Z 438.509,A -85,B 0,C 180,E1 -15947.203,E2 -15947.203} C_VEL
LIN {X 0,Y 310.381,Z 428.01,A -85,B 0,C 180,E1 -15948.823,E2 -15948.823} C_VEL
LIN {X 0,Y 312.103,Z 416.201,A -85,B 0,C 180,E1 -15950.255,E2 -15950.255} C_VEL
LIN {X 0,Y 311.486,Z 406.717,A -85,B 0,C 180,E1 -15951.283,E2 -15951.283} C_VEL
LIN {X 0,Y 309.999,Z 394.793,A -85,B 0,C 180,E1 -15952.378,E2 -15952.378} C_VEL
LIN {X 0,Y 307.694,Z 382.19,A -85,B 0,C 180,E1 -15953.314,E2 -15953.314} C_VEL
LIN {X 0,Y 305.177,Z 371.505,A -85,B 0,C 180,E1 -15953.961,E2 -15953.961} C_VEL
LIN {X 0,Y 305.857,Z 365.459,A -85,B 0,C 180,E1 -15958.101,E2 -15958.101} C_VEL
LIN {X 0,Y 306.599,Z 359.869,A -85,B 0,C 180,E1 -15961.991,E2 -15961.991} C_VEL
LIN {X 0,Y 307.137,Z 355.812,A -85,B 0,C 180,E1 -15964.892,E2 -15964.892} C_VEL
LIN {X 0,Y 307.19,Z 353.226,A -85,B 0,C 180,E1 -15966.799,E2 -15966.799} C_VEL
LIN {X 0,Y 306.881,Z 349.271,A -85,B 0,C 180,E1 -15969.883,E2 -15969.883} C_VEL
LIN {X 0,Y 306.164,Z 344.942,A -85,B 0,C 180,E1 -15973.522,E2 -15973.522} C_VEL
LIN {X 0,Y 305.489,Z 341.434,A -85,B 0,C 180,E1 -15976.801,E2 -15976.801} C_VEL
LIN {X 0,Y 305.454,Z 341.437,A -85,B 0,C 180,E1 -15981.594,E2 -15981.594} C_VEL
LIN {X 0,Y 305.456,Z 341.437,A -85,B 0,C 180,E1 -15984.886,E2 -15984.886} C_VEL
LIN {X 0,Y 305.434,Z 341.441,A -85,B 0,C 180,E1 -15988.357,E2 -15988.357} C_VEL
LIN {X 0,Y 305.468,Z 341.434,A -85,B 0,C 180,E1 -15991.108,E2 -15991.108} C_VEL
LIN {X 0,Y 305.492,Z 341.433,A -85,B 0,C 180,E1 -15994.081,E2 -15994.081} C_VEL
LIN {X 0,Y 305.474,Z 341.436,A -85,B 0,C 180,E1 -15998.401,E2 -15998.401} C_VEL
LIN {X 0,Y 305.581,Z 341.418,A -85,B 0,C 180,E1 -16001.217,E2 -16001.217} C_VEL
LIN {X 0,Y 305.641,Z 341.411,A -85,B 0,C 180,E1 -16005.349,E2 -16005.349} C_VEL
LIN {X 0,Y 305.63,Z 341.412,A -85,B 0,C 180,E1 -16009.399,E2 -16009.399} C_VEL
LIN {X 0,Y 305.806,Z 341.394,A -85,B 0,C 180,E1 -16012.074,E2 -16012.074} C_VEL
LIN {X 0,Y 305.684,Z 341.405,A -85,B 0,C 180,E1 -16014.723,E2 -16014.723} C_VEL
LIN {X 0,Y 305.942,Z 341.373,A -85,B 0,C 180,E1 -16018.684,E2 -16018.684} C_VEL
LIN {X 0,Y 305.941,Z 341.376,A -85,B 0,C 180,E1 -16021.316,E2 -16021.316} C_VEL
LIN {X 0,Y 305.682,Z 341.408,A -85,B 0,C 180,E1 -16025.277,E2 -16025.277} C_VEL
LIN {X 0,Y 305.806,Z 341.391,A -85,B 0,C 180,E1 -16027.926,E2 -16027.926} C_VEL
LIN {X 0,Y 305.594,Z 341.417,A -85,B 0,C 180,E1 -16031.946,E2 -16031.946} C_VEL
LIN {X 0,Y 305.63,Z 341.414,A -85,B 0,C 180,E1 -16035.035,E2 -16035.035} C_VEL
LIN {X 0,Y 305.568,Z 341.422,A -85,B 0,C 180,E1 -16039.445,E2 -16039.445} C_VEL
LIN {X 0,Y 305.479,Z 341.435,A -85,B 0,C 180,E1 -16043.04,E2 -16043.04} C_VEL
LIN {X 0,Y 305.462,Z 341.433,A -85,B 0,C 180,E1 -16046.198,E2 -16046.198} C_VEL
LIN {X 0,Y 305.441,Z 341.44,A -85,B 0,C 180,E1 -16049.034,E2 -16049.034} C_VEL
LIN {X 0,Y 305.43,Z 341.437,A -85,B 0,C 180,E1 -16051.954,E2 -16051.954} C_VEL
LIN {X 0,Y 305.456,Z 341.436,A -85,B 0,C 180,E1 -16055.114,E2 -16055.114} C_VEL
LIN {X 0,Y 305.428,Z 341.441,A -85,B 0,C 180,E1 -16058.526,E2 -16058.526} C_VEL
LIN {X 0,Y 305.431,Z 341.441,A -85,B 0,C 180,E1 -16062.583,E2 -16062.583} C_VEL
LIN {X 0,Y 305.441,Z 341.44,A -85,B 0,C 180,E1 -16066.35,E2 -16066.35} C_VEL
LIN {X 0,Y 305.458,Z 341.437,A -85,B 0,C 180,E1 -16069.894,E2 -16069.894} C_VEL
LIN {X 0,Y 305.457,Z 341.437,A -85,B 0,C 180,E1 -16071.596,E2 -16071.596} C_VEL
LIN {X 0,Y 305.561,Z 343.091,A -85,B 0,C 180,E1 -16073.612,E2 -16073.612} C_VEL
LIN {X 0,Y 305.47,Z 345.76,A -85,B 0,C 180,E1 -16076.485,E2 -16076.485} C_VEL
LIN {X 0,Y 305.212,Z 348.77,A -85,B 0,C 180,E1 -16079.565,E2 -16079.565} C_VEL
LIN {X 0,Y 304.968,Z 351.801,A -85,B 0,C 180,E1 -16082.556,E2 -16082.556} C_VEL
LIN {X 0,Y 304.689,Z 355.532,A -85,B 0,C 180,E1 -16086.075,E2 -16086.075} C_VEL
LIN {X 0,Y 308.524,Z 368.619,A -85,B 0,C 180,E1 -16086.993,E2 -16086.993} C_VEL
LIN {X 0,Y 311.38,Z 380.808,A -85,B 0,C 180,E1 -16088.04,E2 -16088.04} C_VEL
LIN {X 0,Y 313.206,Z 391.542,A -85,B 0,C 180,E1 -16089.133,E2 -16089.133} C_VEL
LIN {X 0,Y 313.272,Z 394.846,A -85,B 0,C 180,E1 -16089.481,E2 -16089.481} C_VEL
LIN {X 0,Y 311.776,Z 406.189,A -85,B 0,C 180,E1 -16090.752,E2 -16090.752} C_VEL
LIN {X 0,Y 310.472,Z 416.634,A -85,B 0,C 180,E1 -16092.247,E2 -16092.247} C_VEL
LIN {X 0,Y 309.076,Z 425.567,A -85,B 0,C 180,E1 -16093.827,E2 -16093.827} C_VEL
LIN {X 0,Y 307.452,Z 434.476,A -85,B 0,C 180,E1 -16095.776,E2 -16095.776} C_VEL
LIN {X 0,Y 306.312,Z 441.64,A -85,B 0,C 180,E1 -16097.748,E2 -16097.748} C_VEL
LIN {X 0,Y 305.455,Z 446.472,A -85,B 0,C 180,E1 -16099.394,E2 -16099.394} C_VEL
LIN {X 0,Y 304.701,Z 451.166,A -85,B 0,C 180,E1 -16101.378,E2 -16101.378} C_VEL
LIN {X 0,Y 304.261,Z 454.754,A -85,B 0,C 180,E1 -16103.369,E2 -16103.369} C_VEL
LIN {X 0,Y 304.038,Z 456.608,A -85,B 0,C 180,E1 -16104.695,E2 -16104.695} C_VEL
LIN {X 0,Y 303.87,Z 458.002,A -85,B 0,C 180,E1 -16106.022,E2 -16106.022} C_VEL
LIN {X 0,Y 303.628,Z 459.606,A -85,B 0,C 180,E1 -16108.674,E2 -16108.674} C_VEL
LIN {X 0,Y 303.613,Z 459.836,A -85,B 0,C 180,E1 -16110.001,E2 -16110.001} C_VEL
LIN {X 0,Y 303.628,Z 459.644,A -85,B 0,C 180,E1 -16111.327,E2 -16111.327} C_VEL
LIN {X 0,Y 303.869,Z 458.089,A -85,B 0,C 180,E1 -16113.979,E2 -16113.979} C_VEL
LIN {X 0,Y 304.038,Z 456.733,A -85,B 0,C 180,E1 -16115.306,E2 -16115.306} C_VEL
LIN {X 0,Y 304.374,Z 453.974,A -85,B 0,C 180,E1 -16117.23,E2 -16117.23} C_VEL
LIN {X 0,Y 304.857,Z 449.984,A -85,B 0,C 180,E1 -16119.287,E2 -16119.287} C_VEL
LIN {X 0,Y 305.737,Z 444.967,A -85,B 0,C 180,E1 -16121.268,E2 -16121.268} C_VEL
LIN {X 0,Y 306.792,Z 438.649,A -85,B 0,C 180,E1 -16123.243,E2 -16123.243} C_VEL
LIN {X 0,Y 308.156,Z 430.74,A -85,B 0,C 180,E1 -16125.205,E2 -16125.205} C_VEL
LIN {X 0,Y 309.811,Z 420.9,A -85,B 0,C 180,E1 -16127.152,E2 -16127.152} C_VEL
LIN {X 0,Y 311.191,Z 410.573,A -85,B 0,C 180,E1 -16128.774,E2 -16128.774} C_VEL
LIN {X 0,Y 312.585,Z 400.337,A -85,B 0,C 180,E1 -16130.052,E2 -16130.052} C_VEL
LIN {X 0,Y 313.371,Z 392.659,A -85,B 0,C 180,E1 -16130.857,E2 -16130.857} C_VEL
LIN {X 0,Y 311.487,Z 381.365,A -85,B 0,C 180,E1 -16132.021,E2 -16132.021} C_VEL
LIN {X 0,Y 308.615,Z 368.842,A -85,B 0,C 180,E1 -16133.101,E2 -16133.101} C_VEL
LIN {X 0,Y 304.665,Z 355.494,A -85,B 0,C 180,E1 -16134.08,E2 -16134.08} C_VEL
LIN {X 0,Y 304.94,Z 351.923,A -85,B 0,C 180,E1 -16137.448,E2 -16137.448} C_VEL
LIN {X 0,Y 305.21,Z 348.914,A -85,B 0,C 180,E1 -16140.437,E2 -16140.437} C_VEL
LIN {X 0,Y 305.513,Z 345.34,A -85,B 0,C 180,E1 -16144.091,E2 -16144.091} C_VEL
LIN {X 0,Y 305.552,Z 342.887,A -85,B 0,C 180,E1 -16146.728,E2 -16146.728} C_VEL
LIN {X 0,Y 305.422,Z 341.442,A -85,B 0,C 180,E1 -16148.522,E2 -16148.522} C_VEL
LIN {X 0,Y 305.441,Z 341.442,A -85,B 0,C 180,E1 -16151.857,E2 -16151.857} C_VEL
LIN {X 0,Y 305.398,Z 341.446,A -85,B 0,C 180,E1 -16155.511,E2 -16155.511} C_VEL
LIN {X 0,Y 305.41,Z 341.441,A -85,B 0,C 180,E1 -16158.138,E2 -16158.138} C_VEL
LIN {X 0,Y 305.445,Z 341.439,A -85,B 0,C 180,E1 -16161.593,E2 -16161.593} C_VEL
LIN {X 0,Y 305.461,Z 341.435,A -85,B 0,C 180,E1 -16164.886,E2 -16164.886} C_VEL
LIN {X 0,Y 305.44,Z 341.435,A -85,B 0,C 180,E1 -16168.358,E2 -16168.358} C_VEL
LIN {X 0,Y 305.473,Z 341.435,A -85,B 0,C 180,E1 -16171.109,E2 -16171.109} C_VEL
LIN {X 0,Y 305.498,Z 341.428,A -85,B 0,C 180,E1 -16174.081,E2 -16174.081} C_VEL
LIN {X 0,Y 305.478,Z 341.432,A -85,B 0,C 180,E1 -16178.401,E2 -16178.401} C_VEL
LIN {X 0,Y 305.587,Z 341.42,A -85,B 0,C 180,E1 -16181.217,E2 -16181.217} C_VEL
LIN {X 0,Y 305.642,Z 341.411,A -85,B 0,C 180,E1 -16185.397,E2 -16185.397} C_VEL
LIN {X 0,Y 304.927,Z 341.503,A -85,B 0,C 180,E1 -16186.496,E2 -16186.496} C_VEL
LIN {X 0,Y 302.15,Z 341.847,A -85,B 0,C 180,E1 -16188.29,E2 -16188.29} C_VEL
LIN {X 0,Y 299.836,Z 342.137,A -85,B 0,C 180,E1 -16189.744,E2 -16189.744} C_VEL
LIN {X 0,Y 298.84,Z 342.261,A -85,B 0,C 180,E1 -16190.868,E2 -16190.868} C_VEL
LIN {X 0,Y 298.755,Z 342.269,A -85,B 0,C 180,E1 -16191.248,E2 -16191.248} C_VEL
LIN {X 0,Y 298.796,Z 342.263,A -85,B 0,C 180,E1 -16193.246,E2 -16193.246} C_VEL
LIN {X 0,Y 298.914,Z 342.251,A -85,B 0,C 180,E1 -16198.653,E2 -16198.653} C_VEL
LIN {X 0,Y 298.913,Z 342.248,A -85,B 0,C 180,E1 -16201.347,E2 -16201.347} C_VEL
LIN {X 0,Y 298.785,Z 342.266,A -85,B 0,C 180,E1 -16206.754,E2 -16206.754} C_VEL
LIN {X 0,Y 298.633,Z 342.285,A -85,B 0,C 180,E1 -16209.482,E2 -16209.482} C_VEL
LIN {X 0,Y 298.549,Z 342.297,A -85,B 0,C 180,E1 -16213.615,E2 -16213.615} C_VEL
LIN {X 0,Y 298.546,Z 342.297,A -85,B 0,C 180,E1 -16216.409,E2 -16216.409} C_VEL
LIN {X 0,Y 298.508,Z 342.304,A -85,B 0,C 180,E1 -16219.654,E2 -16219.654} C_VEL
LIN {X 0,Y 298.421,Z 342.315,A -85,B 0,C 180,E1 -16223.601,E2 -16223.601} C_VEL
LIN {X 0,Y 298.406,Z 342.313,A -85,B 0,C 180,E1 -16226.582,E2 -16226.582} C_VEL
LIN {X 0,Y 298.391,Z 342.319,A -85,B 0,C 180,E1 -16229.644,E2 -16229.644} C_VEL
LIN {X 0,Y 298.391,Z 342.316,A -85,B 0,C 180,E1 -16232.801,E2 -16232.801} C_VEL
LIN {X 0,Y 298.427,Z 342.312,A -85,B 0,C 180,E1 -16236.803,E2 -16236.803} C_VEL
LIN {X 0,Y 298.372,Z 342.319,A -85,B 0,C 180,E1 -16239.492,E2 -16239.492} C_VEL
LIN {X 0,Y 298.418,Z 342.343,A -85,B 0,C 180,E1 -16242.846,E2 -16242.846} C_VEL
LIN {X 0,Y 299.234,Z 346.944,A -85,B 0,C 180,E1 -16247.07,E2 -16247.07} C_VEL
LIN {X 0,Y 299.927,Z 351.3,A -85,B 0,C 180,E1 -16250.753,E2 -16250.753} C_VEL
LIN {X 0,Y 300.178,Z 355.647,A -85,B 0,C 180,E1 -16254.175,E2 -16254.175} C_VEL
LIN {X 0,Y 299.625,Z 360.275,A -85,B 0,C 180,E1 -16257.61,E2 -16257.61} C_VEL
LIN {X 0,Y 298.939,Z 365.276,A -85,B 0,C 180,E1 -16261.187,E2 -16261.187} C_VEL
LIN {X 0,Y 298.173,Z 371.27,A -85,B 0,C 180,E1 -16265.42,E2 -16265.42} C_VEL
LIN {X 0,Y 301.396,Z 384.822,A -85,B 0,C 180,E1 -16266.301,E2 -16266.301} C_VEL
LIN {X 0,Y 303.518,Z 397.154,A -85,B 0,C 180,E1 -16267.301,E2 -16267.301} C_VEL
LIN {X 0,Y 304.802,Z 407.893,A -85,B 0,C 180,E1 -16268.351,E2 -16268.351} C_VEL
LIN {X 0,Y 305.37,Z 416.096,A -85,B 0,C 180,E1 -16269.277,E2 -16269.277} C_VEL
LIN {X 0,Y 303.9,Z 426.713,A -85,B 0,C 180,E1 -16270.583,E2 -16270.583} C_VEL
LIN {X 0,Y 302.401,Z 436.418,A -85,B 0,C 180,E1 -16272.065,E2 -16272.065} C_VEL
LIN {X 0,Y 301.03,Z 445.265,A -85,B 0,C 180,E1 -16273.73,E2 -16273.73} C_VEL
LIN {X 0,Y 299.542,Z 453.889,A -85,B 0,C 180,E1 -16275.738,E2 -16275.738} C_VEL
LIN {X 0,Y 298.339,Z 460.786,A -85,B 0,C 180,E1 -16277.759,E2 -16277.759} C_VEL
LIN {X 0,Y 297.545,Z 466.319,A -85,B 0,C 180,E1 -16279.796,E2 -16279.796} C_VEL
LIN {X 0,Y 296.995,Z 470.661,A -85,B 0,C 180,E1 -16281.837,E2 -16281.837} C_VEL
LIN {X 0,Y 296.631,Z 474.521,A -85,B 0,C 180,E1 -16284.324,E2 -16284.324} C_VEL
LIN {X 0,Y 296.548,Z 476.226,A -85,B 0,C 180,E1 -16285.922,E2 -16285.922} C_VEL
LIN {X 0,Y 296.536,Z 477.225,A -85,B 0,C 180,E1 -16287.283,E2 -16287.283} C_VEL
LIN {X 0,Y 296.481,Z 477.834,A -85,B 0,C 180,E1 -16288.641,E2 -16288.641} C_VEL
LIN {X 0,Y 296.487,Z 478.049,A -85,B 0,C 180,E1 -16289.999,E2 -16289.999} C_VEL
LIN {X 0,Y 296.481,Z 477.83,A -85,B 0,C 180,E1 -16291.358,E2 -16291.358} C_VEL
LIN {X 0,Y 296.536,Z 477.22,A -85,B 0,C 180,E1 -16292.716,E2 -16292.716} C_VEL
LIN {X 0,Y 296.547,Z 476.218,A -85,B 0,C 180,E1 -16294.076,E2 -16294.076} C_VEL
LIN {X 0,Y 296.623,Z 474.528,A -85,B 0,C 180,E1 -16295.66,E2 -16295.66} C_VEL
LIN {X 0,Y 296.981,Z 470.637,A -85,B 0,C 180,E1 -16298.162,E2 -16298.162} C_VEL
LIN {X 0,Y 297.546,Z 466.287,A -85,B 0,C 180,E1 -16300.203,E2 -16300.203} C_VEL
LIN {X 0,Y 298.338,Z 460.747,A -85,B 0,C 180,E1 -16302.24,E2 -16302.24} C_VEL
LIN {X 0,Y 299.547,Z 453.84,A -85,B 0,C 180,E1 -16304.261,E2 -16304.261} C_VEL
LIN {X 0,Y 300.733,Z 446.788,A -85,B 0,C 180,E1 -16305.937,E2 -16305.937} C_VEL
LIN {X 0,Y 302.084,Z 438.29,A -85,B 0,C 180,E1 -16307.604,E2 -16307.604} C_VEL
LIN {X 0,Y 303.664,Z 427.791,A -85,B 0,C 180,E1 -16309.256,E2 -16309.256} C_VEL
LIN {X 0,Y 305.245,Z 417.411,A -85,B 0,C 180,E1 -16310.555,E2 -16310.555} C_VEL
LIN {X 0,Y 305.031,Z 411.231,A -85,B 0,C 180,E1 -16311.276,E2 -16311.276} C_VEL
LIN {X 0,Y 303.862,Z 399.609,A -85,B 0,C 180,E1 -16312.461,E2 -16312.461} C_VEL
LIN {X 0,Y 301.697,Z 386.328,A -85,B 0,C 180,E1 -16313.566,E2 -16313.566} C_VEL
LIN {X 0,Y 298.64,Z 373.59,A -85,B 0,C 180,E1 -16314.435,E2 -16314.435} C_VEL
LIN {X 0,Y 298.171,Z 371.263,A -85,B 0,C 180,E1 -16314.566,E2 -16314.566} C_VEL
LIN {X 0,Y 298.936,Z 365.251,A -85,B 0,C 180,E1 -16318.812,E2 -16318.812} C_VEL
LIN {X 0,Y 299.665,Z 359.914,A -85,B 0,C 180,E1 -16322.642,E2 -16322.642} C_VEL
LIN {X 0,Y 300.192,Z 355.619,A -85,B 0,C 180,E1 -16325.822,E2 -16325.822} C_VEL
LIN {X 0,Y 299.962,Z 351.124,A -85,B 0,C 180,E1 -16329.36,E2 -16329.36} C_VEL
LIN {X 0,Y 299.234,Z 346.504,A -85,B 0,C 180,E1 -16333.274,E2 -16333.274} C_VEL
LIN {X 0,Y 298.431,Z 342.312,A -85,B 0,C 180,E1 -16337.156,E2 -16337.156} C_VEL
LIN {X 0,Y 298.379,Z 342.321,A -85,B 0,C 180,E1 -16341.01,E2 -16341.01} C_VEL
LIN {X 0,Y 298.399,Z 342.315,A -85,B 0,C 180,E1 -16343.927,E2 -16343.927} C_VEL
LIN {X 0,Y 298.386,Z 342.317,A -85,B 0,C 180,E1 -16347.199,E2 -16347.199} C_VEL
LIN {X 0,Y 298.394,Z 342.318,A -85,B 0,C 180,E1 -16350.624,E2 -16350.624} C_VEL
LIN {X 0,Y 298.436,Z 342.31,A -85,B 0,C 180,E1 -16354.92,E2 -16354.92} C_VEL
LIN {X 0,Y 298.432,Z 342.309,A -85,B 0,C 180,E1 -16359.314,E2 -16359.314} C_VEL
LIN {X 0,Y 298.529,Z 342.301,A -85,B 0,C 180,E1 -16362.179,E2 -16362.179} C_VEL
LIN {X 0,Y 298.585,Z 342.29,A -85,B 0,C 180,E1 -16364.994,E2 -16364.994} C_VEL
LIN {X 0,Y 298.585,Z 342.289,A -85,B 0,C 180,E1 -16369.146,E2 -16369.146} C_VEL
LIN {X 0,Y 298.751,Z 342.273,A -85,B 0,C 180,E1 -16371.886,E2 -16371.886} C_VEL
LIN {X 0,Y 298.655,Z 342.281,A -85,B 0,C 180,E1 -16374.599,E2 -16374.599} C_VEL
LIN {X 0,Y 298.909,Z 342.249,A -85,B 0,C 180,E1 -16378.653,E2 -16378.653} C_VEL
LIN {X 0,Y 298.909,Z 342.252,A -85,B 0,C 180,E1 -16381.347,E2 -16381.347} C_VEL
